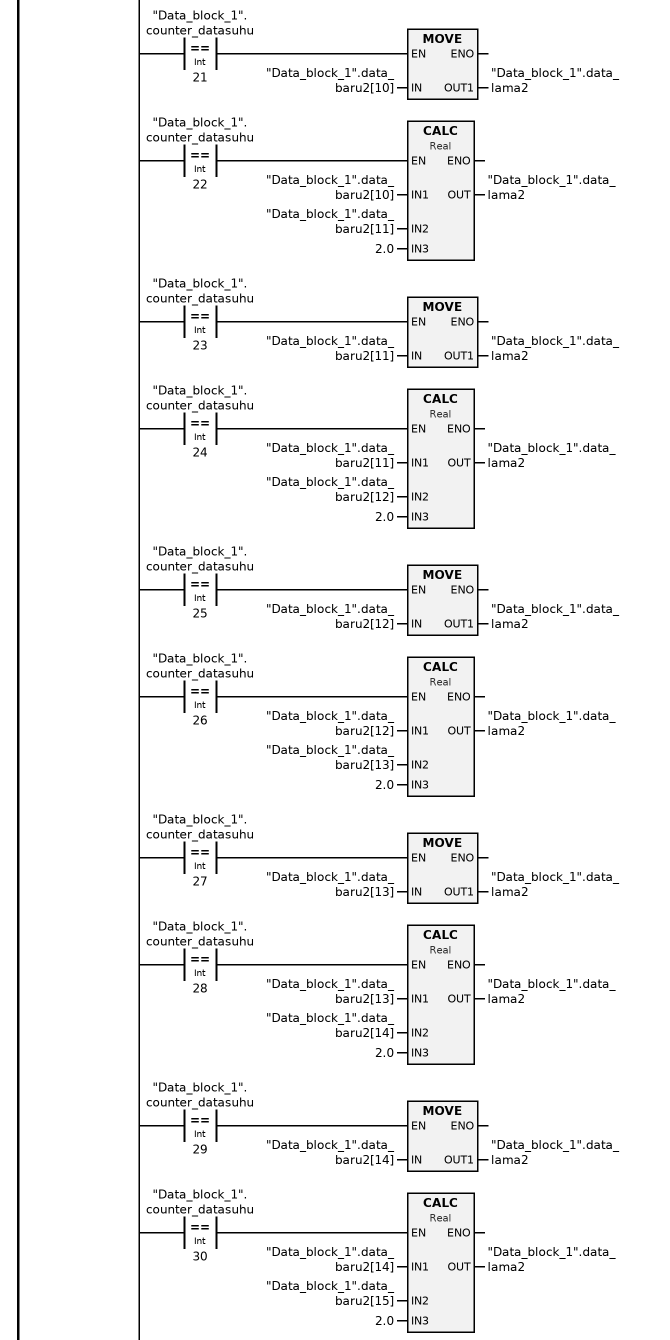
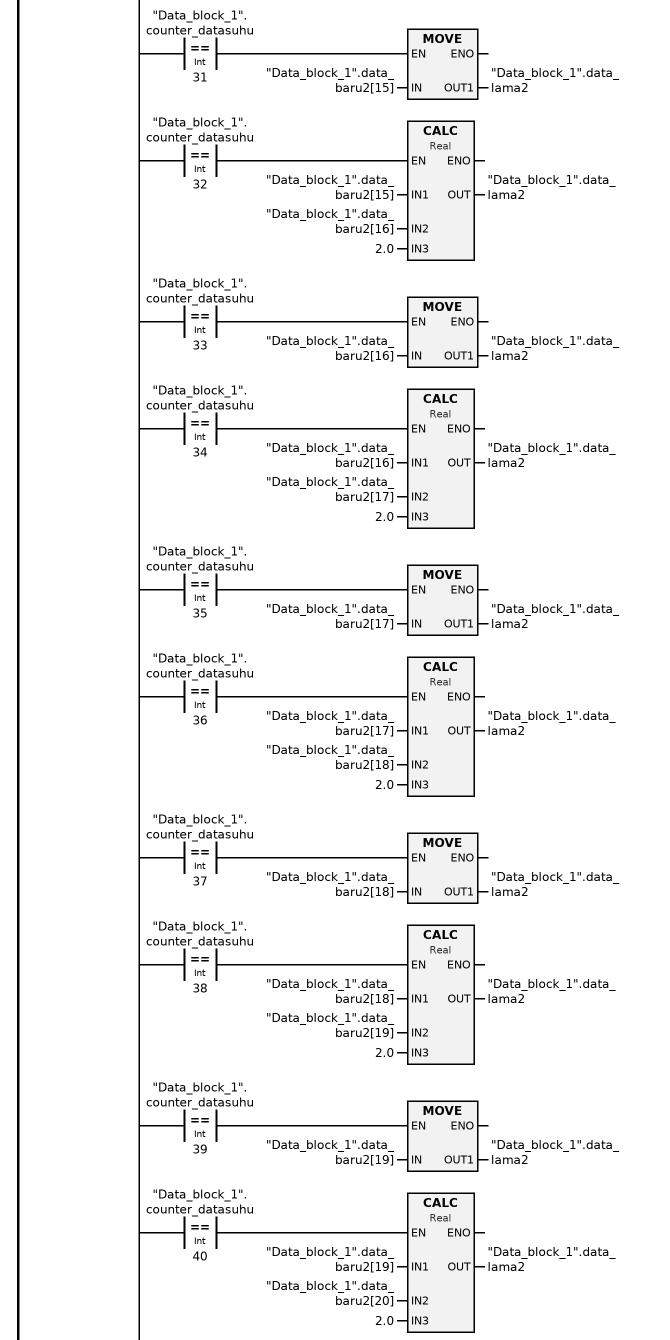
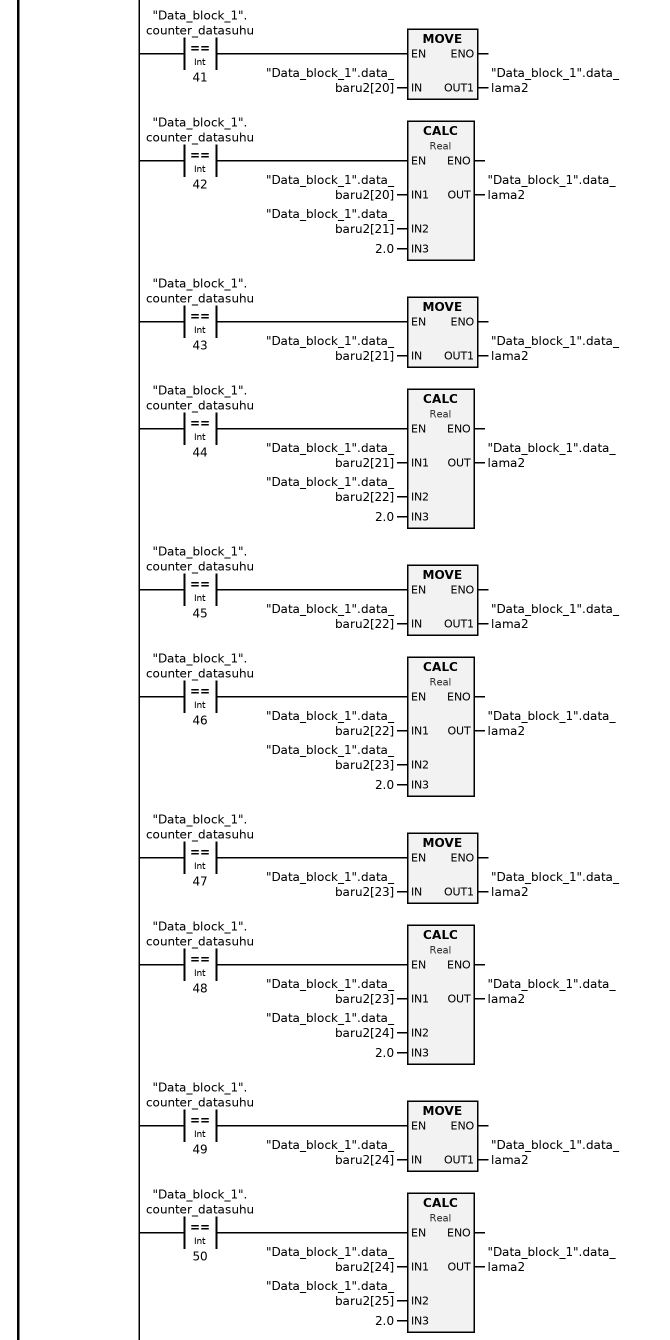
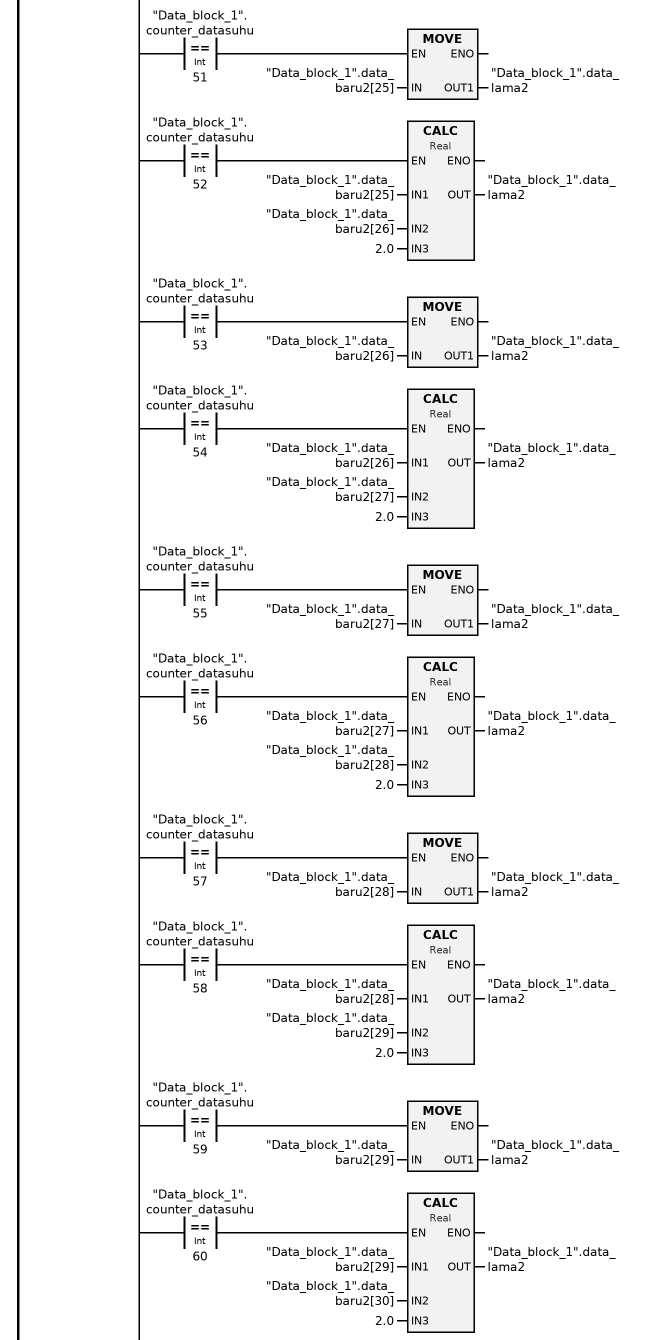
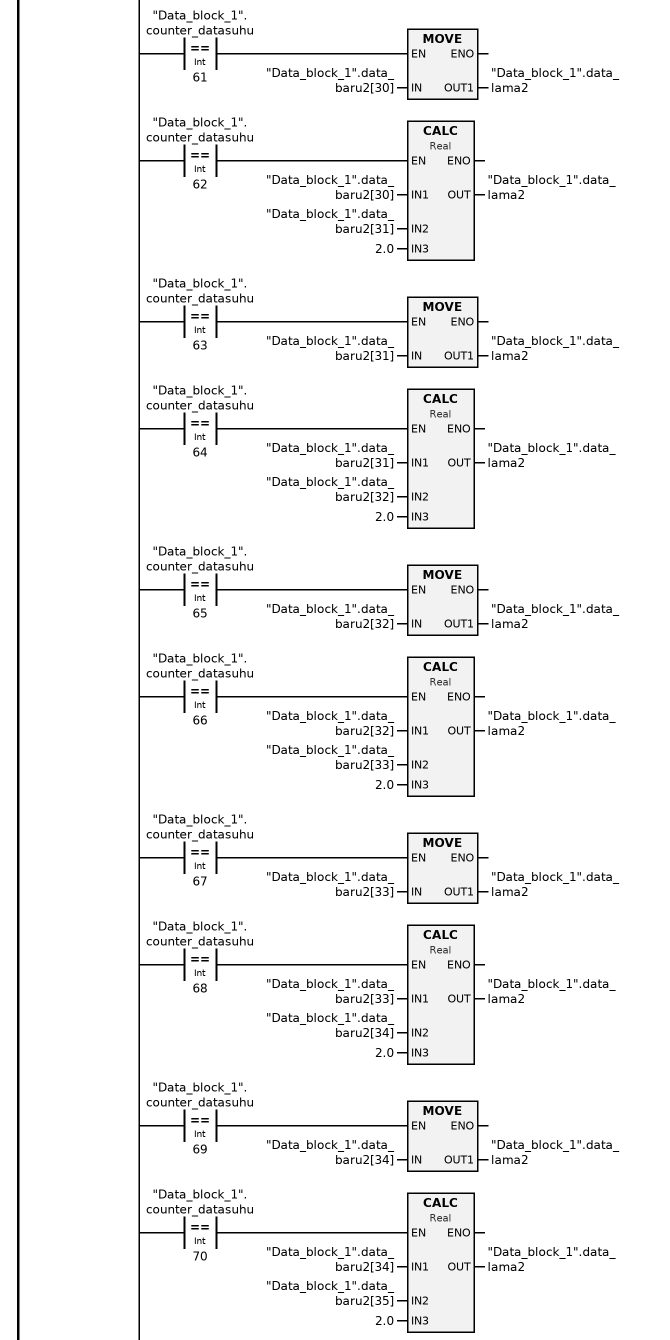
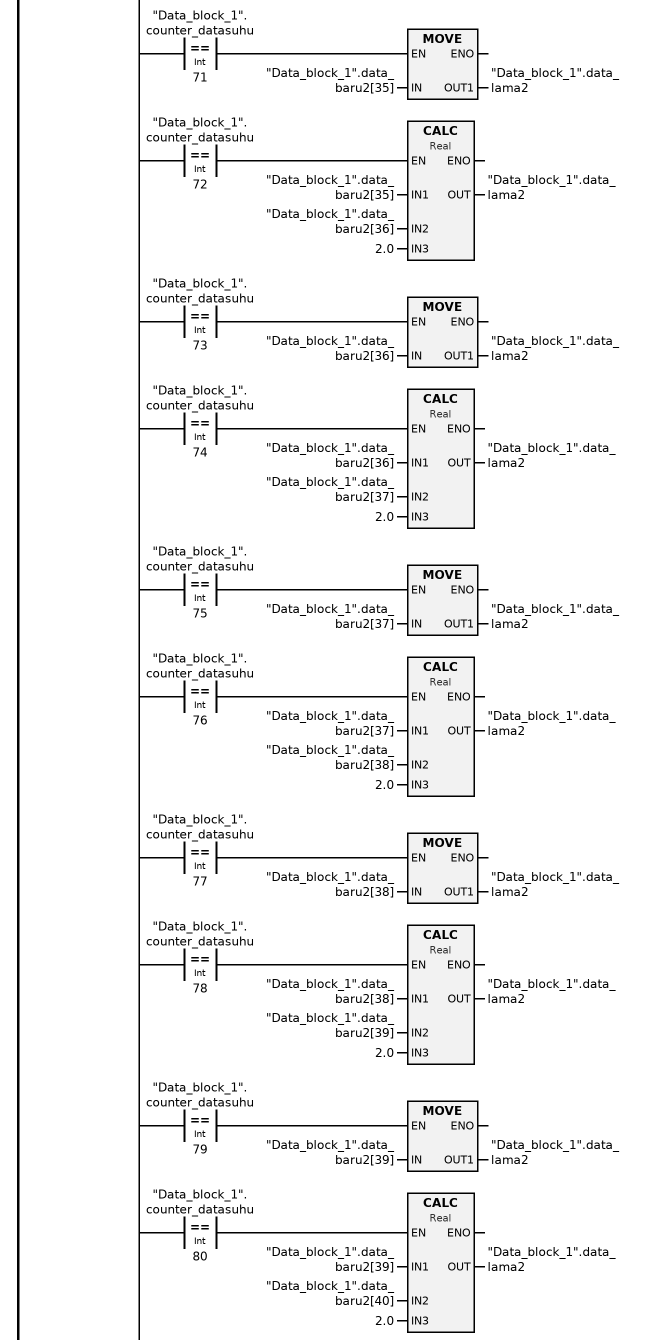
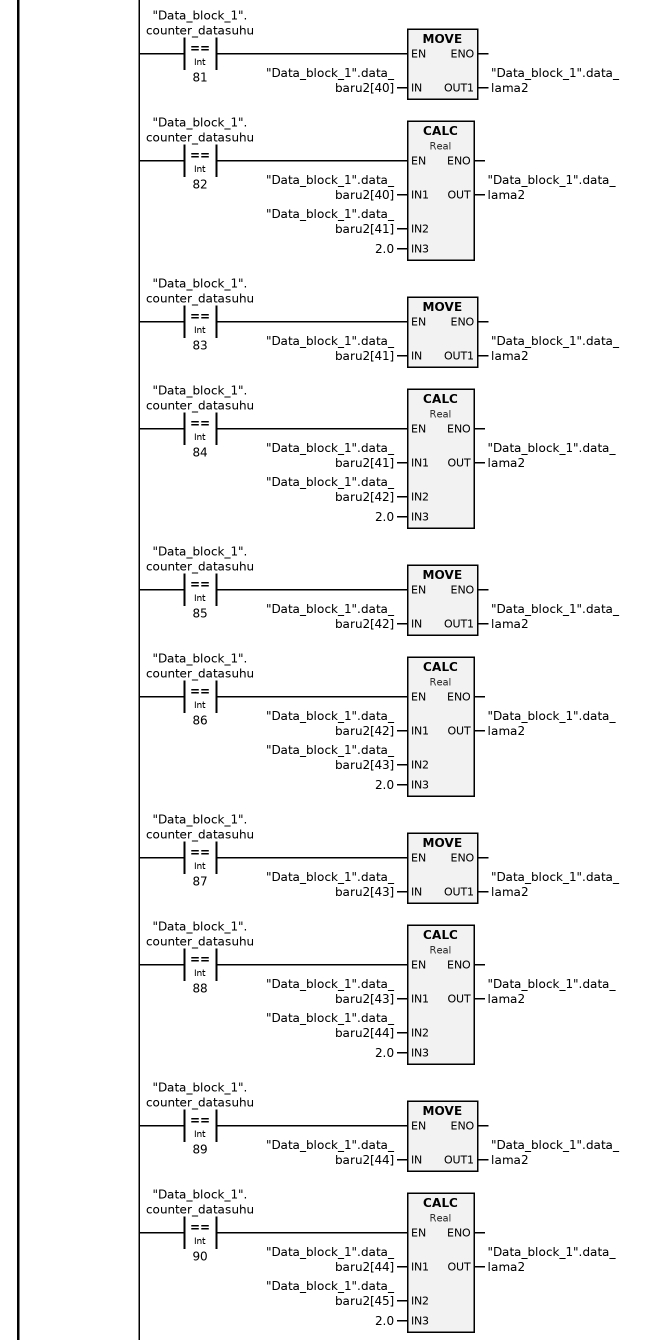
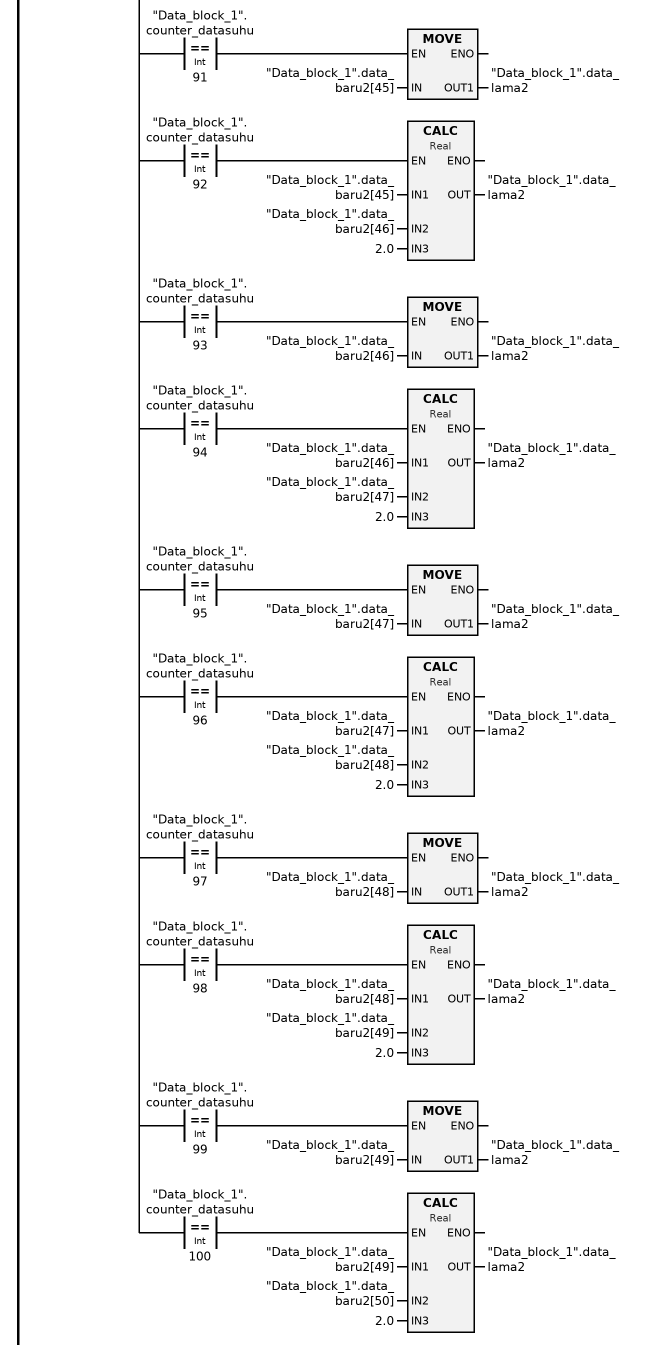
   #_w1 := NOT "Data_block_1".Lock_A;
   IF #_w1 AND ("Data_block_1".counter_datasuhu = 1) THEN
       "Data_block_1".data_lama2 := "Data_block_1".data_baru2[0];
   END_IF;
   IF #_w1 AND ("Data_block_1".counter_datasuhu = 2) THEN
       CALC(in1 := "Data_block_1".data_baru2[0],
            in2 := "Data_block_1".data_baru2[1],
            in3 := 2.0,
            out => "Data_block_1".data_lama2);
   END_IF;
   IF #_w1 AND ("Data_block_1".counter_datasuhu = 3) THEN
       "Data_block_1".data_lama2 := "Data_block_1".data_baru2[1];
   END_IF;
   IF #_w1 AND ("Data_block_1".counter_datasuhu = 4) THEN
       CALC(in1 := "Data_block_1".data_baru2[1],
            in2 := "Data_block_1".data_baru2[2],
            in3 := 2.0,
            out => "Data_block_1".data_lama2);
   END_IF;
   IF #_w1 AND ("Data_block_1".counter_datasuhu = 5) THEN
       "Data_block_1".data_lama2 := "Data_block_1".data_baru2[2];
   END_IF;
   IF #_w1 AND ("Data_block_1".counter_datasuhu = 6) THEN
       CALC(in1 := "Data_block_1".data_baru2[2],
            in2 := "Data_block_1".data_baru2[3],
            in3 := 2.0,
            out => "Data_block_1".data_lama2);
   END_IF;
   IF #_w1 AND ("Data_block_1".counter_datasuhu = 7) THEN
       "Data_block_1".data_lama2 := "Data_block_1".data_baru2[3];
   END_IF;
   IF #_w1 AND ("Data_block_1".counter_datasuhu = 8) THEN
       CALC(in1 := "Data_block_1".data_baru2[3],
            in2 := "Data_block_1".data_baru2[4],
            in3 := 2.0,
            out => "Data_block_1".data_lama2);
   END_IF;
   IF #_w1 AND ("Data_block_1".counter_datasuhu = 9) THEN
       "Data_block_1".data_lama2 := "Data_block_1".data_baru2[4];
   END_IF;
   IF #_w1 AND ("Data_block_1".counter_datasuhu = 10) THEN
       CALC(in1 := "Data_block_1".data_baru2[4],
            in2 := "Data_block_1".data_baru2[5],
            in3 := 2.0,
            out => "Data_block_1".data_lama2);
   END_IF;
   IF #_w1 AND ("Data_block_1".counter_datasuhu = 11) THEN
       "Data_block_1".data_lama2 := "Data_block_1".data_baru2[5];
   END_IF;
   IF #_w1 AND ("Data_block_1".counter_datasuhu = 12) THEN
       CALC(in1 := "Data_block_1".data_baru2[5],
            in2 := "Data_block_1".data_baru2[6],
            in3 := 2.0,
            out => "Data_block_1".data_lama2);
   END_IF;
   IF #_w1 AND ("Data_block_1".counter_datasuhu = 13) THEN
       "Data_block_1".data_lama2 := "Data_block_1".data_baru2[6];
   END_IF;
   IF #_w1 AND ("Data_block_1".counter_datasuhu = 14) THEN
       CALC(in1 := "Data_block_1".data_baru2[6],
            in2 := "Data_block_1".data_baru2[7],
            in3 := 2.0,
            out => "Data_block_1".data_lama2);
   END_IF;
   IF #_w1 AND ("Data_block_1".counter_datasuhu = 15) THEN
       "Data_block_1".data_lama2 := "Data_block_1".data_baru2[7];
   END_IF;
   IF #_w1 AND ("Data_block_1".counter_datasuhu = 16) THEN
       CALC(in1 := "Data_block_1".data_baru2[7],
            in2 := "Data_block_1".data_baru2[8],
            in3 := 2.0,
            out => "Data_block_1".data_lama2);
   END_IF;
   IF #_w1 AND ("Data_block_1".counter_datasuhu = 17) THEN
       "Data_block_1".data_lama2 := "Data_block_1".data_baru2[8];
   END_IF;
   IF #_w1 AND ("Data_block_1".counter_datasuhu = 18) THEN
       CALC(in1 := "Data_block_1".data_baru2[8],
            in2 := "Data_block_1".data_baru2[9],
            in3 := 2.0,
            out => "Data_block_1".data_lama2);
   END_IF;
   IF #_w1 AND ("Data_block_1".counter_datasuhu = 19) THEN
       "Data_block_1".data_lama2 := "Data_block_1".data_baru2[9];
   END_IF;
   IF #_w1 AND ("Data_block_1".counter_datasuhu = 20) THEN
       CALC(in1 := "Data_block_1".data_baru2[9],
            in2 := "Data_block_1".data_baru2[10],
            in3 := 2.0,
            out => "Data_block_1".data_lama2);
   END_IF;
   IF #_w1 AND ("Data_block_1".counter_datasuhu = 21) THEN
       "Data_block_1".data_lama2 := "Data_block_1".data_baru2[10];
   END_IF;
   IF #_w1 AND ("Data_block_1".counter_datasuhu = 22) THEN
       CALC(in1 := "Data_block_1".data_baru2[10],
            in2 := "Data_block_1".data_baru2[11],
            in3 := 2.0,
            out => "Data_block_1".data_lama2);
   END_IF;
   IF #_w1 AND ("Data_block_1".counter_datasuhu = 23) THEN
       "Data_block_1".data_lama2 := "Data_block_1".data_baru2[11];
   END_IF;
   IF #_w1 AND ("Data_block_1".counter_datasuhu = 24) THEN
       CALC(in1 := "Data_block_1".data_baru2[11],
            in2 := "Data_block_1".data_baru2[12],
            in3 := 2.0,
            out => "Data_block_1".data_lama2);
   END_IF;
   IF #_w1 AND ("Data_block_1".counter_datasuhu = 25) THEN
       "Data_block_1".data_lama2 := "Data_block_1".data_baru2[12];
   END_IF;
   IF #_w1 AND ("Data_block_1".counter_datasuhu = 26) THEN
       CALC(in1 := "Data_block_1".data_baru2[12],
            in2 := "Data_block_1".data_baru2[13],
            in3 := 2.0,
            out => "Data_block_1".data_lama2);
   END_IF;
   IF #_w1 AND ("Data_block_1".counter_datasuhu = 27) THEN
       "Data_block_1".data_lama2 := "Data_block_1".data_baru2[13];
   END_IF;
   IF #_w1 AND ("Data_block_1".counter_datasuhu = 28) THEN
       CALC(in1 := "Data_block_1".data_baru2[13],
            in2 := "Data_block_1".data_baru2[14],
            in3 := 2.0,
            out => "Data_block_1".data_lama2);
   END_IF;
   IF #_w1 AND ("Data_block_1".counter_datasuhu = 29) THEN
       "Data_block_1".data_lama2 := "Data_block_1".data_baru2[14];
   END_IF;
   IF #_w1 AND ("Data_block_1".counter_datasuhu = 30) THEN
       CALC(in1 := "Data_block_1".data_baru2[14],
            in2 := "Data_block_1".data_baru2[15],
            in3 := 2.0,
            out => "Data_block_1".data_lama2);
   END_IF;
   IF #_w1 AND ("Data_block_1".counter_datasuhu = 31) THEN
       "Data_block_1".data_lama2 := "Data_block_1".data_baru2[15];
   END_IF;
   IF #_w1 AND ("Data_block_1".counter_datasuhu = 32) THEN
       CALC(in1 := "Data_block_1".data_baru2[15],
            in2 := "Data_block_1".data_baru2[16],
            in3 := 2.0,
            out => "Data_block_1".data_lama2);
   END_IF;
   IF #_w1 AND ("Data_block_1".counter_datasuhu = 33) THEN
       "Data_block_1".data_lama2 := "Data_block_1".data_baru2[16];
   END_IF;
   IF #_w1 AND ("Data_block_1".counter_datasuhu = 34) THEN
       CALC(in1 := "Data_block_1".data_baru2[16],
            in2 := "Data_block_1".data_baru2[17],
            in3 := 2.0,
            out => "Data_block_1".data_lama2);
   END_IF;
   IF #_w1 AND ("Data_block_1".counter_datasuhu = 35) THEN
       "Data_block_1".data_lama2 := "Data_block_1".data_baru2[17];
   END_IF;
   IF #_w1 AND ("Data_block_1".counter_datasuhu = 36) THEN
       CALC(in1 := "Data_block_1".data_baru2[17],
            in2 := "Data_block_1".data_baru2[18],
            in3 := 2.0,
            out => "Data_block_1".data_lama2);
   END_IF;
   IF #_w1 AND ("Data_block_1".counter_datasuhu = 37) THEN
       "Data_block_1".data_lama2 := "Data_block_1".data_baru2[18];
   END_IF;
   IF #_w1 AND ("Data_block_1".counter_datasuhu = 38) THEN
       CALC(in1 := "Data_block_1".data_baru2[18],
            in2 := "Data_block_1".data_baru2[19],
            in3 := 2.0,
            out => "Data_block_1".data_lama2);
   END_IF;
   IF #_w1 AND ("Data_block_1".counter_datasuhu = 39) THEN
       "Data_block_1".data_lama2 := "Data_block_1".data_baru2[19];
   END_IF;
   IF #_w1 AND ("Data_block_1".counter_datasuhu = 40) THEN
       CALC(in1 := "Data_block_1".data_baru2[19],
            in2 := "Data_block_1".data_baru2[20],
            in3 := 2.0,
            out => "Data_block_1".data_lama2);
   END_IF;
   IF #_w1 AND ("Data_block_1".counter_datasuhu = 41) THEN
       "Data_block_1".data_lama2 := "Data_block_1".data_baru2[20];
   END_IF;
   IF #_w1 AND ("Data_block_1".counter_datasuhu = 42) THEN
       CALC(in1 := "Data_block_1".data_baru2[20],
            in2 := "Data_block_1".data_baru2[21],
            in3 := 2.0,
            out => "Data_block_1".data_lama2);
   END_IF;
   IF #_w1 AND ("Data_block_1".counter_datasuhu = 43) THEN
       "Data_block_1".data_lama2 := "Data_block_1".data_baru2[21];
   END_IF;
   IF #_w1 AND ("Data_block_1".counter_datasuhu = 44) THEN
       CALC(in1 := "Data_block_1".data_baru2[21],
            in2 := "Data_block_1".data_baru2[22],
            in3 := 2.0,
            out => "Data_block_1".data_lama2);
   END_IF;
   IF #_w1 AND ("Data_block_1".counter_datasuhu = 45) THEN
       "Data_block_1".data_lama2 := "Data_block_1".data_baru2[22];
   END_IF;
   IF #_w1 AND ("Data_block_1".counter_datasuhu = 46) THEN
       CALC(in1 := "Data_block_1".data_baru2[22],
            in2 := "Data_block_1".data_baru2[23],
            in3 := 2.0,
            out => "Data_block_1".data_lama2);
   END_IF;
   IF #_w1 AND ("Data_block_1".counter_datasuhu = 47) THEN
       "Data_block_1".data_lama2 := "Data_block_1".data_baru2[23];
   END_IF;
   IF #_w1 AND ("Data_block_1".counter_datasuhu = 48) THEN
       CALC(in1 := "Data_block_1".data_baru2[23],
            in2 := "Data_block_1".data_baru2[24],
            in3 := 2.0,
            out => "Data_block_1".data_lama2);
   END_IF;
   IF #_w1 AND ("Data_block_1".counter_datasuhu = 49) THEN
       "Data_block_1".data_lama2 := "Data_block_1".data_baru2[24];
   END_IF;
   IF #_w1 AND ("Data_block_1".counter_datasuhu = 50) THEN
       CALC(in1 := "Data_block_1".data_baru2[24],
            in2 := "Data_block_1".data_baru2[25],
            in3 := 2.0,
            out => "Data_block_1".data_lama2);
   END_IF;
   IF #_w1 AND ("Data_block_1".counter_datasuhu = 51) THEN
       "Data_block_1".data_lama2 := "Data_block_1".data_baru2[25];
   END_IF;
   IF #_w1 AND ("Data_block_1".counter_datasuhu = 52) THEN
       CALC(in1 := "Data_block_1".data_baru2[25],
            in2 := "Data_block_1".data_baru2[26],
            in3 := 2.0,
            out => "Data_block_1".data_lama2);
   END_IF;
   IF #_w1 AND ("Data_block_1".counter_datasuhu = 53) THEN
       "Data_block_1".data_lama2 := "Data_block_1".data_baru2[26];
   END_IF;
   IF #_w1 AND ("Data_block_1".counter_datasuhu = 54) THEN
       CALC(in1 := "Data_block_1".data_baru2[26],
            in2 := "Data_block_1".data_baru2[27],
            in3 := 2.0,
            out => "Data_block_1".data_lama2);
   END_IF;
   IF #_w1 AND ("Data_block_1".counter_datasuhu = 55) THEN
       "Data_block_1".data_lama2 := "Data_block_1".data_baru2[27];
   END_IF;
   IF #_w1 AND ("Data_block_1".counter_datasuhu = 56) THEN
       CALC(in1 := "Data_block_1".data_baru2[27],
            in2 := "Data_block_1".data_baru2[28],
            in3 := 2.0,
            out => "Data_block_1".data_lama2);
   END_IF;
   IF #_w1 AND ("Data_block_1".counter_datasuhu = 57) THEN
       "Data_block_1".data_lama2 := "Data_block_1".data_baru2[28];
   END_IF;
   IF #_w1 AND ("Data_block_1".counter_datasuhu = 58) THEN
       CALC(in1 := "Data_block_1".data_baru2[28],
            in2 := "Data_block_1".data_baru2[29],
            in3 := 2.0,
            out => "Data_block_1".data_lama2);
   END_IF;
   IF #_w1 AND ("Data_block_1".counter_datasuhu = 59) THEN
       "Data_block_1".data_lama2 := "Data_block_1".data_baru2[29];
   END_IF;
   IF #_w1 AND ("Data_block_1".counter_datasuhu = 60) THEN
       CALC(in1 := "Data_block_1".data_baru2[29],
            in2 := "Data_block_1".data_baru2[30],
            in3 := 2.0,
            out => "Data_block_1".data_lama2);
   END_IF;
   IF #_w1 AND ("Data_block_1".counter_datasuhu = 61) THEN
       "Data_block_1".data_lama2 := "Data_block_1".data_baru2[30];
   END_IF;
   IF #_w1 AND ("Data_block_1".counter_datasuhu = 62) THEN
       CALC(in1 := "Data_block_1".data_baru2[30],
            in2 := "Data_block_1".data_baru2[31],
            in3 := 2.0,
            out => "Data_block_1".data_lama2);
   END_IF;
   IF #_w1 AND ("Data_block_1".counter_datasuhu = 63) THEN
       "Data_block_1".data_lama2 := "Data_block_1".data_baru2[31];
   END_IF;
   IF #_w1 AND ("Data_block_1".counter_datasuhu = 64) THEN
       CALC(in1 := "Data_block_1".data_baru2[31],
            in2 := "Data_block_1".data_baru2[32],
            in3 := 2.0,
            out => "Data_block_1".data_lama2);
   END_IF;
   IF #_w1 AND ("Data_block_1".counter_datasuhu = 65) THEN
       "Data_block_1".data_lama2 := "Data_block_1".data_baru2[32];
   END_IF;
   IF #_w1 AND ("Data_block_1".counter_datasuhu = 66) THEN
       CALC(in1 := "Data_block_1".data_baru2[32],
            in2 := "Data_block_1".data_baru2[33],
            in3 := 2.0,
            out => "Data_block_1".data_lama2);
   END_IF;
   IF #_w1 AND ("Data_block_1".counter_datasuhu = 67) THEN
       "Data_block_1".data_lama2 := "Data_block_1".data_baru2[33];
   END_IF;
   IF #_w1 AND ("Data_block_1".counter_datasuhu = 68) THEN
       CALC(in1 := "Data_block_1".data_baru2[33],
            in2 := "Data_block_1".data_baru2[34],
            in3 := 2.0,
            out => "Data_block_1".data_lama2);
   END_IF;
   IF #_w1 AND ("Data_block_1".counter_datasuhu = 69) THEN
       "Data_block_1".data_lama2 := "Data_block_1".data_baru2[34];
   END_IF;
   IF #_w1 AND ("Data_block_1".counter_datasuhu = 70) THEN
       CALC(in1 := "Data_block_1".data_baru2[34],
            in2 := "Data_block_1".data_baru2[35],
            in3 := 2.0,
            out => "Data_block_1".data_lama2);
   END_IF;
   IF #_w1 AND ("Data_block_1".counter_datasuhu = 71) THEN
       "Data_block_1".data_lama2 := "Data_block_1".data_baru2[35];
   END_IF;
   IF #_w1 AND ("Data_block_1".counter_datasuhu = 72) THEN
       CALC(in1 := "Data_block_1".data_baru2[35],
            in2 := "Data_block_1".data_baru2[36],
            in3 := 2.0,
            out => "Data_block_1".data_lama2);
   END_IF;
   IF #_w1 AND ("Data_block_1".counter_datasuhu = 73) THEN
       "Data_block_1".data_lama2 := "Data_block_1".data_baru2[36];
   END_IF;
   IF #_w1 AND ("Data_block_1".counter_datasuhu = 74) THEN
       CALC(in1 := "Data_block_1".data_baru2[36],
            in2 := "Data_block_1".data_baru2[37],
            in3 := 2.0,
            out => "Data_block_1".data_lama2);
   END_IF;
   IF #_w1 AND ("Data_block_1".counter_datasuhu = 75) THEN
       "Data_block_1".data_lama2 := "Data_block_1".data_baru2[37];
   END_IF;
   IF #_w1 AND ("Data_block_1".counter_datasuhu = 76) THEN
       CALC(in1 := "Data_block_1".data_baru2[37],
            in2 := "Data_block_1".data_baru2[38],
            in3 := 2.0,
            out => "Data_block_1".data_lama2);
   END_IF;
   IF #_w1 AND ("Data_block_1".counter_datasuhu = 77) THEN
       "Data_block_1".data_lama2 := "Data_block_1".data_baru2[38];
   END_IF;
   IF #_w1 AND ("Data_block_1".counter_datasuhu = 78) THEN
       CALC(in1 := "Data_block_1".data_baru2[38],
            in2 := "Data_block_1".data_baru2[39],
            in3 := 2.0,
            out => "Data_block_1".data_lama2);
   END_IF;
   IF #_w1 AND ("Data_block_1".counter_datasuhu = 79) THEN
       "Data_block_1".data_lama2 := "Data_block_1".data_baru2[39];
   END_IF;
   IF #_w1 AND ("Data_block_1".counter_datasuhu = 80) THEN
       CALC(in1 := "Data_block_1".data_baru2[39],
            in2 := "Data_block_1".data_baru2[40],
            in3 := 2.0,
            out => "Data_block_1".data_lama2);
   END_IF;
   IF #_w1 AND ("Data_block_1".counter_datasuhu = 81) THEN
       "Data_block_1".data_lama2 := "Data_block_1".data_baru2[40];
   END_IF;
   IF #_w1 AND ("Data_block_1".counter_datasuhu = 82) THEN
       CALC(in1 := "Data_block_1".data_baru2[40],
            in2 := "Data_block_1".data_baru2[41],
            in3 := 2.0,
            out => "Data_block_1".data_lama2);
   END_IF;
   IF #_w1 AND ("Data_block_1".counter_datasuhu = 83) THEN
       "Data_block_1".data_lama2 := "Data_block_1".data_baru2[41];
   END_IF;
   IF #_w1 AND ("Data_block_1".counter_datasuhu = 84) THEN
       CALC(in1 := "Data_block_1".data_baru2[41],
            in2 := "Data_block_1".data_baru2[42],
            in3 := 2.0,
            out => "Data_block_1".data_lama2);
   END_IF;
   IF #_w1 AND ("Data_block_1".counter_datasuhu = 85) THEN
       "Data_block_1".data_lama2 := "Data_block_1".data_baru2[42];
   END_IF;
   IF #_w1 AND ("Data_block_1".counter_datasuhu = 86) THEN
       CALC(in1 := "Data_block_1".data_baru2[42],
            in2 := "Data_block_1".data_baru2[43],
            in3 := 2.0,
            out => "Data_block_1".data_lama2);
   END_IF;
   IF #_w1 AND ("Data_block_1".counter_datasuhu = 87) THEN
       "Data_block_1".data_lama2 := "Data_block_1".data_baru2[43];
   END_IF;
   IF #_w1 AND ("Data_block_1".counter_datasuhu = 88) THEN
       CALC(in1 := "Data_block_1".data_baru2[43],
            in2 := "Data_block_1".data_baru2[44],
            in3 := 2.0,
            out => "Data_block_1".data_lama2);
   END_IF;
   IF #_w1 AND ("Data_block_1".counter_datasuhu = 89) THEN
       "Data_block_1".data_lama2 := "Data_block_1".data_baru2[44];
   END_IF;
   IF #_w1 AND ("Data_block_1".counter_datasuhu = 90) THEN
       CALC(in1 := "Data_block_1".data_baru2[44],
            in2 := "Data_block_1".data_baru2[45],
            in3 := 2.0,
            out => "Data_block_1".data_lama2);
   END_IF;
   IF #_w1 AND ("Data_block_1".counter_datasuhu = 91) THEN
       "Data_block_1".data_lama2 := "Data_block_1".data_baru2[45];
   END_IF;
   IF #_w1 AND ("Data_block_1".counter_datasuhu = 92) THEN
       CALC(in1 := "Data_block_1".data_baru2[45],
            in2 := "Data_block_1".data_baru2[46],
            in3 := 2.0,
            out => "Data_block_1".data_lama2);
   END_IF;
   IF #_w1 AND ("Data_block_1".counter_datasuhu = 93) THEN
       "Data_block_1".data_lama2 := "Data_block_1".data_baru2[46];
   END_IF;
   IF #_w1 AND ("Data_block_1".counter_datasuhu = 94) THEN
       CALC(in1 := "Data_block_1".data_baru2[46],
            in2 := "Data_block_1".data_baru2[47],
            in3 := 2.0,
            out => "Data_block_1".data_lama2);
   END_IF;
   IF #_w1 AND ("Data_block_1".counter_datasuhu = 95) THEN
       "Data_block_1".data_lama2 := "Data_block_1".data_baru2[47];
   END_IF;
   IF #_w1 AND ("Data_block_1".counter_datasuhu = 96) THEN
       CALC(in1 := "Data_block_1".data_baru2[47],
            in2 := "Data_block_1".data_baru2[48],
            in3 := 2.0,
            out => "Data_block_1".data_lama2);
   END_IF;
   IF #_w1 AND ("Data_block_1".counter_datasuhu = 97) THEN
       "Data_block_1".data_lama2 := "Data_block_1".data_baru2[48];
   END_IF;
   IF #_w1 AND ("Data_block_1".counter_datasuhu = 98) THEN
       CALC(in1 := "Data_block_1".data_baru2[48],
            in2 := "Data_block_1".data_baru2[49],
            in3 := 2.0,
            out => "Data_block_1".data_lama2);
   END_IF;
   IF #_w1 AND ("Data_block_1".counter_datasuhu = 99) THEN
       "Data_block_1".data_lama2 := "Data_block_1".data_baru2[49];
   END_IF;
   IF #_w1 AND ("Data_block_1".counter_datasuhu = 100) THEN
       CALC(in1 := "Data_block_1".data_baru2[49],
            in2 := "Data_block_1".data_baru2[50],
            in3 := 2.0,
            out => "Data_block_1".data_lama2);
   END_IF;
END_REGION

REGION Network 29: Memasukkan Data
   // ketika pemutus aktif dan counter bertambah, data suhu lama dipindahkan ke array dataroda (dari 0-37) serta sarana akan ditampilkan pada tabel sesuai roda pertama tiap sarana
   // ketika pemutus aktif, data suhu, data suhu lama , dan data suhu baru akan menjadi 0
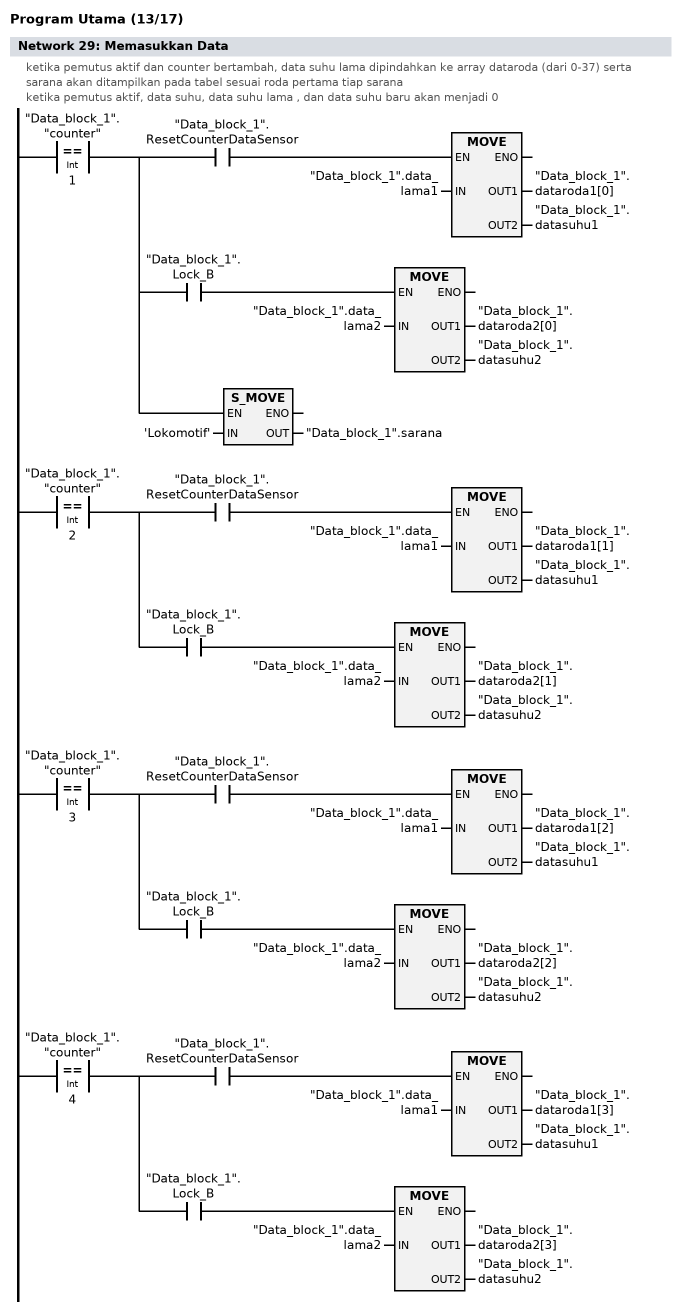
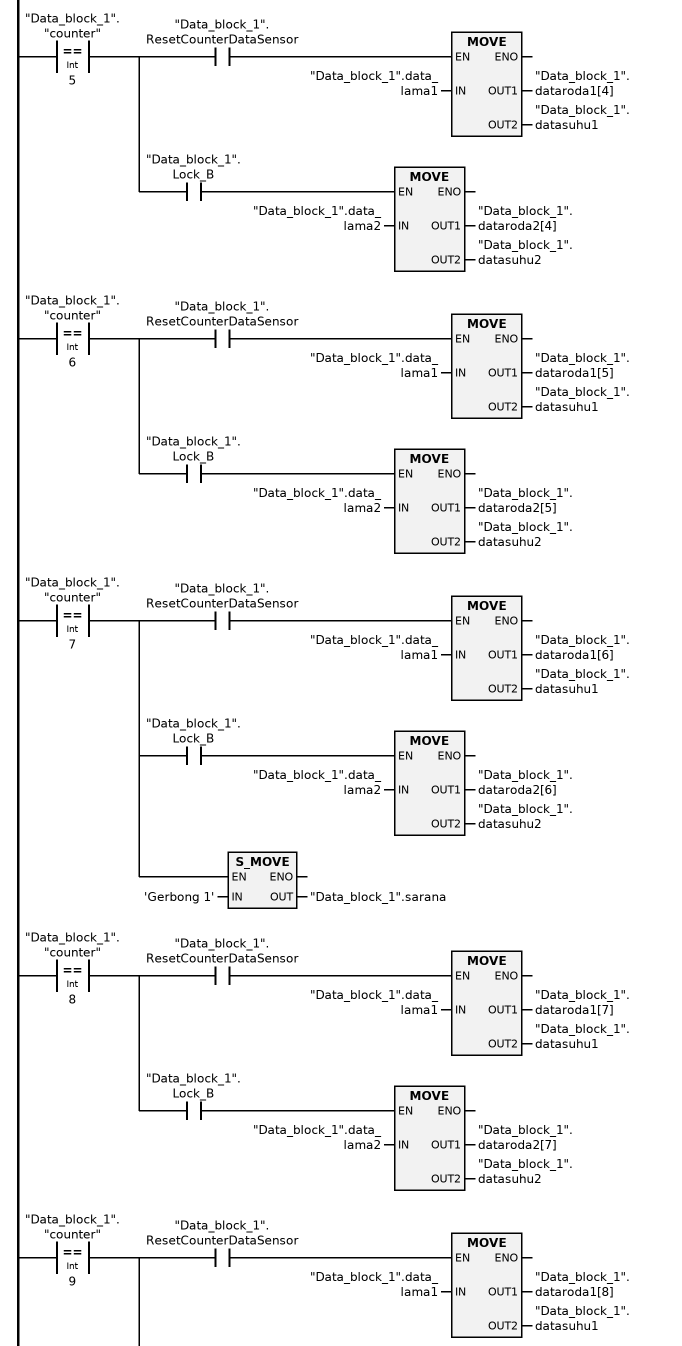
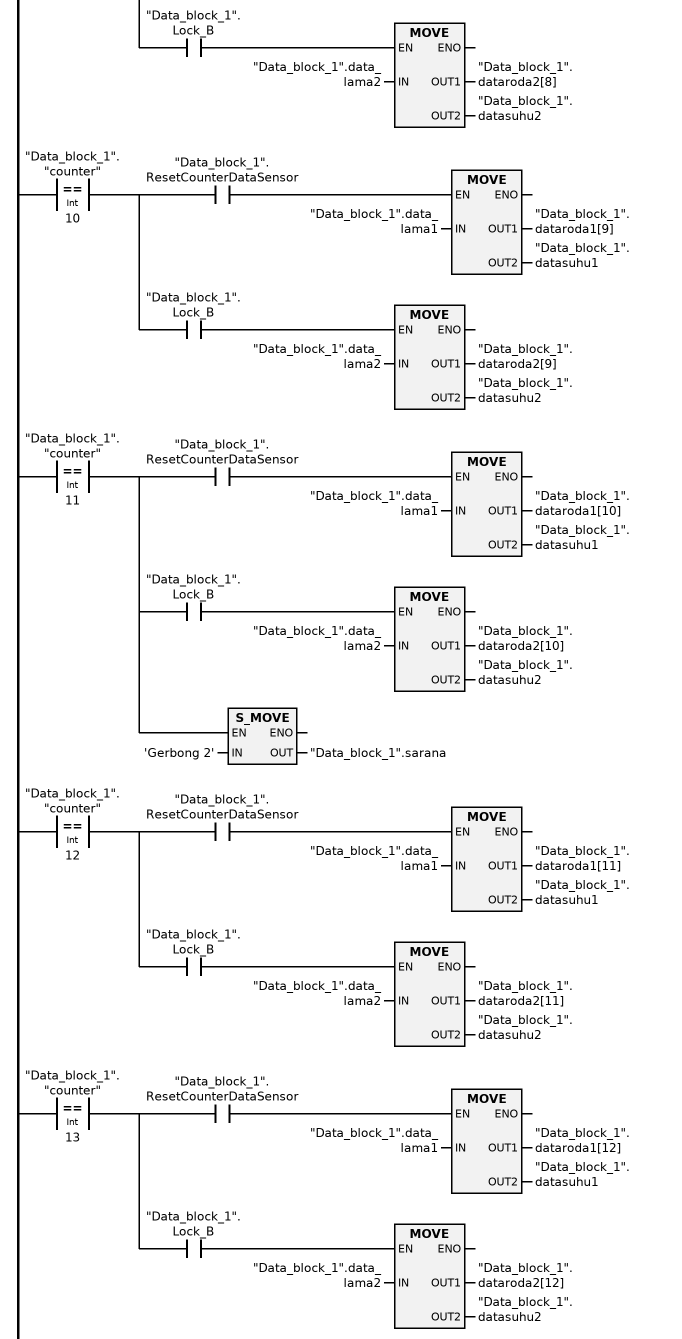
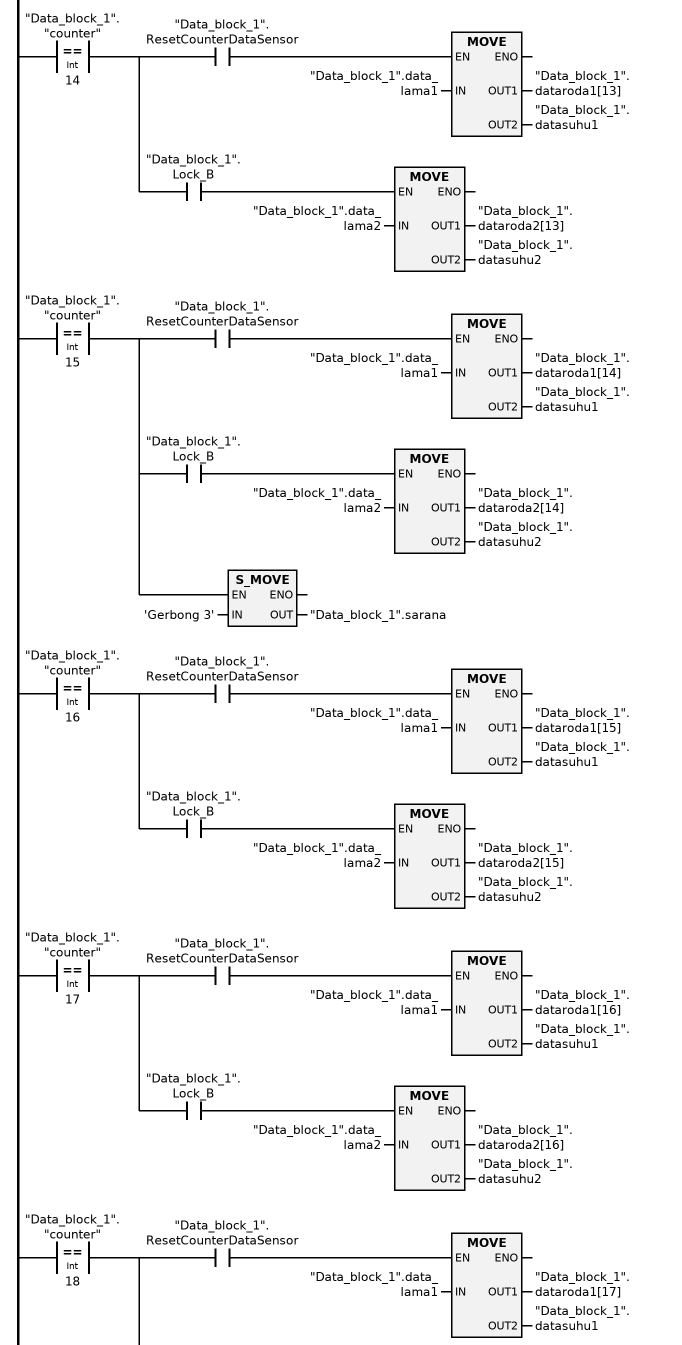
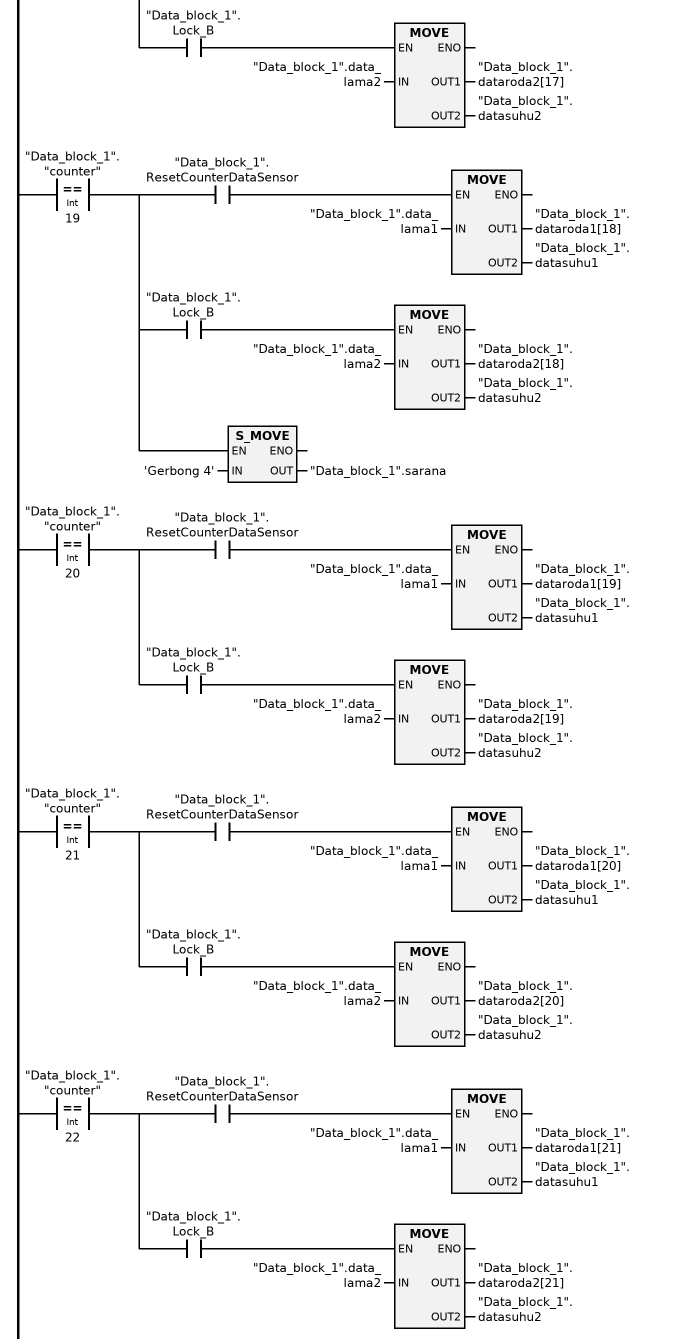
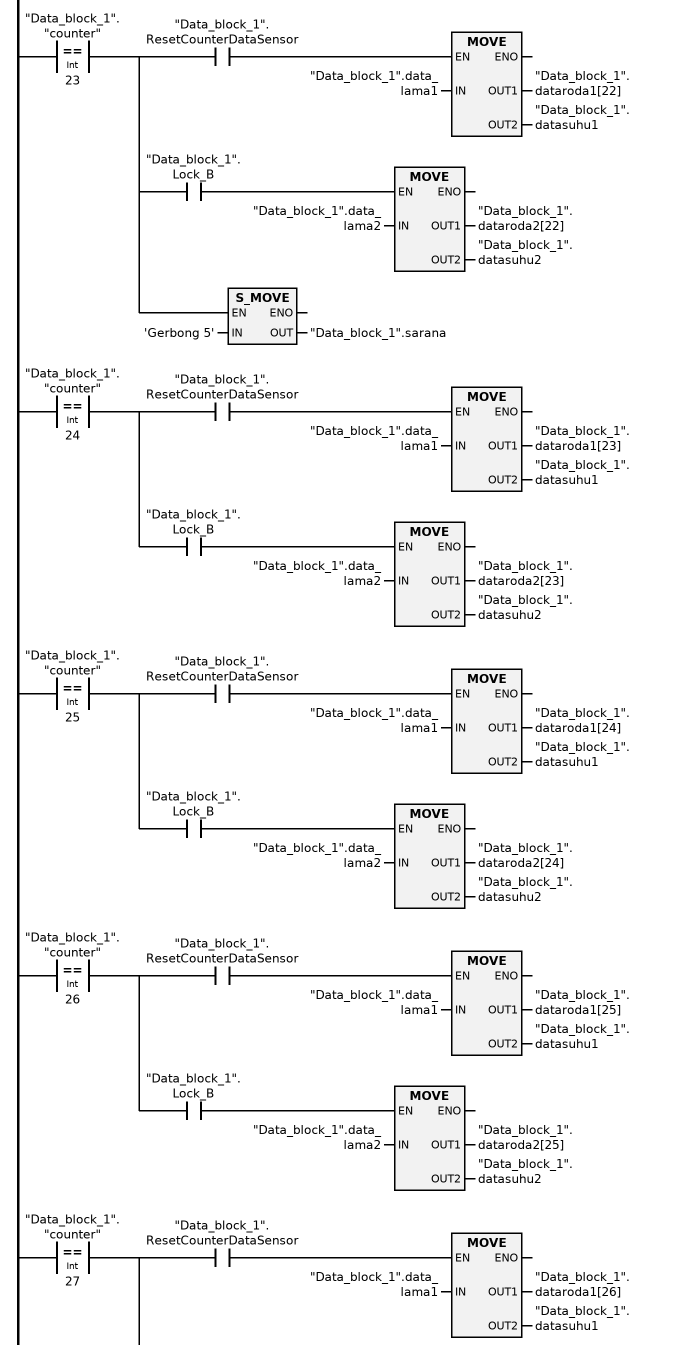
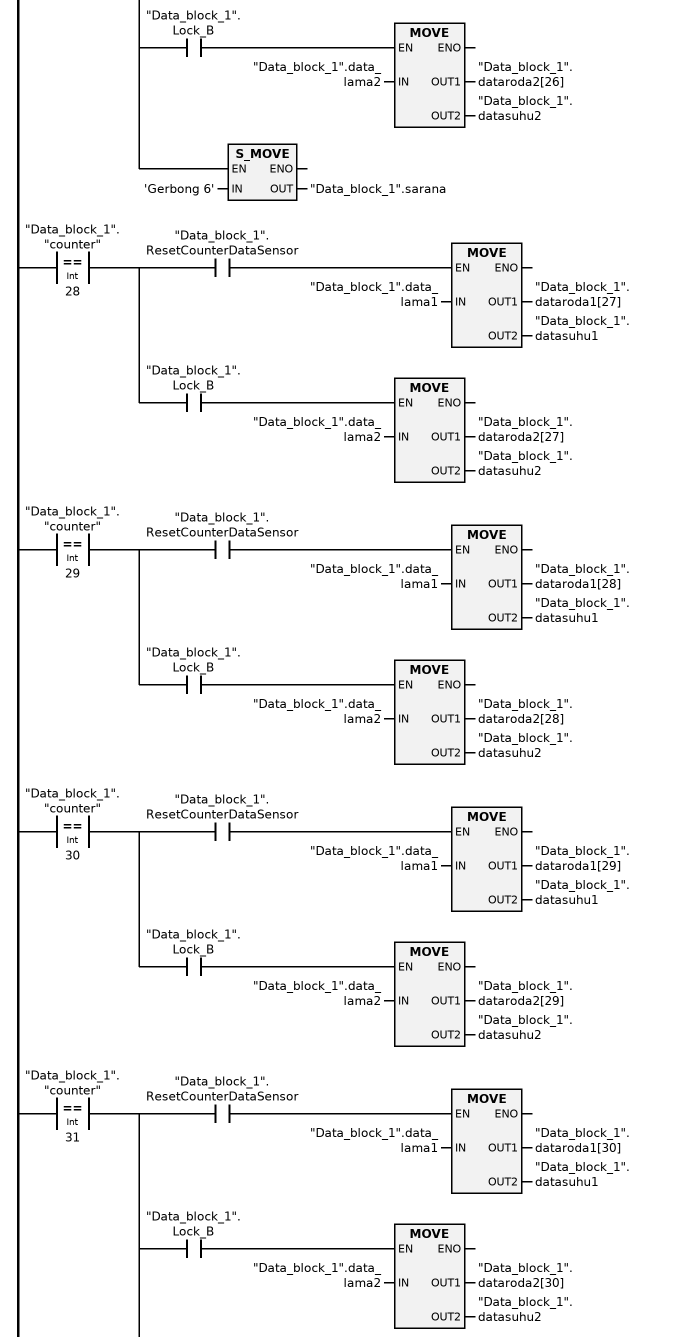
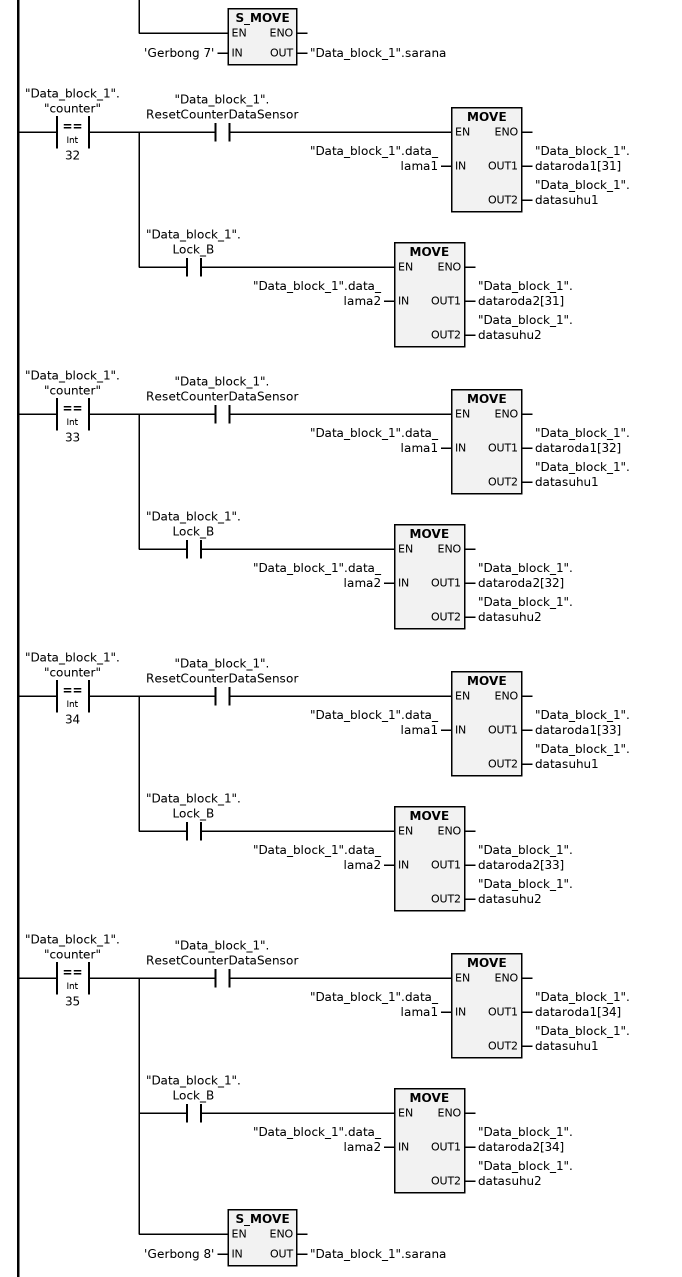
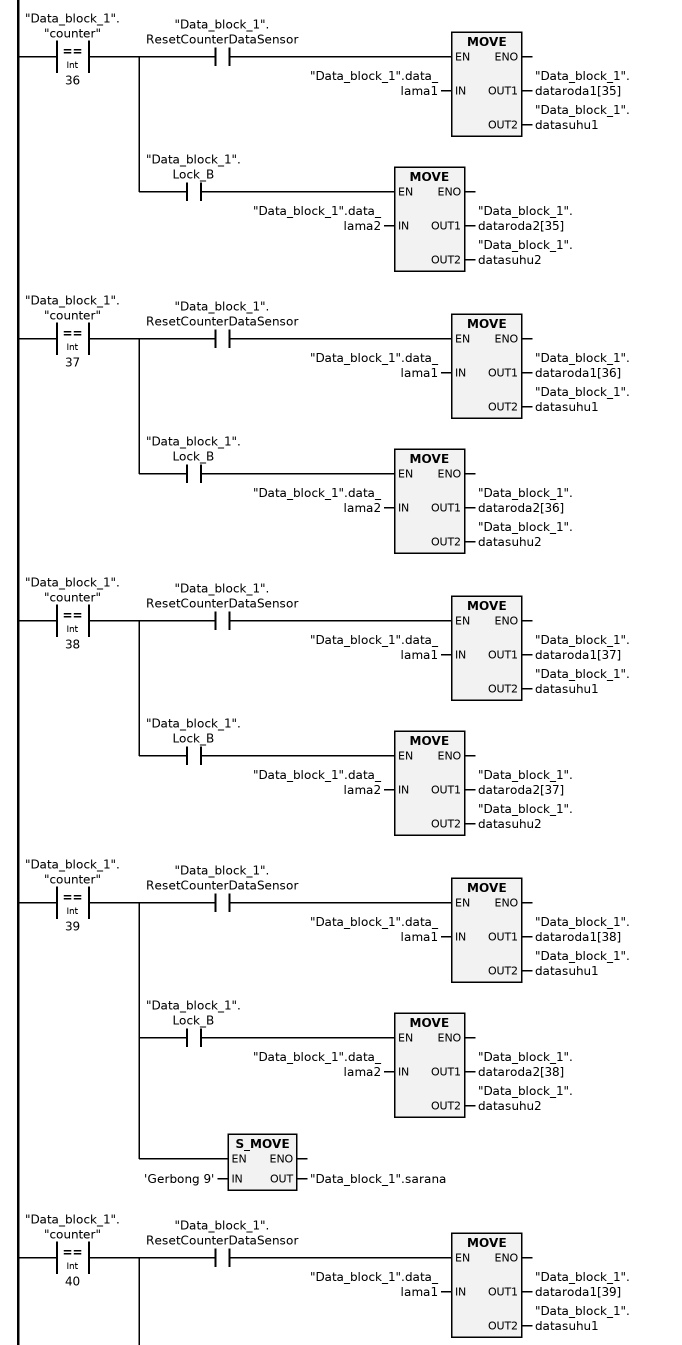
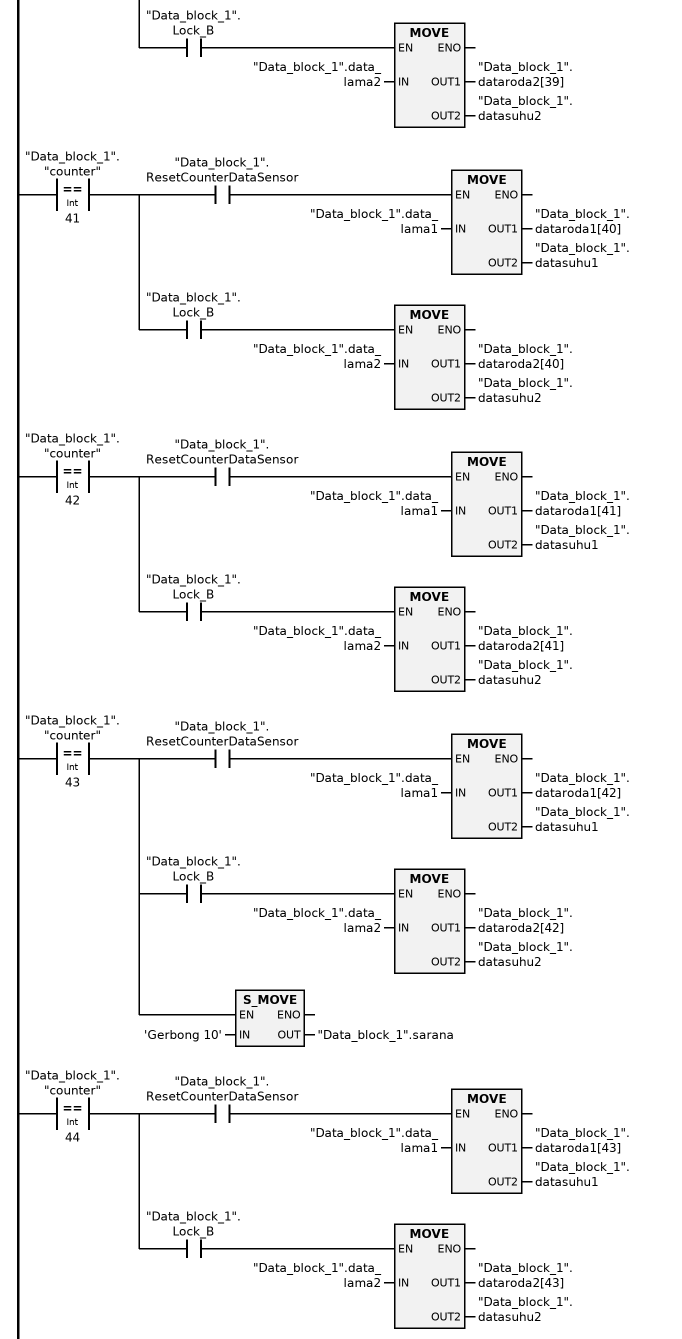
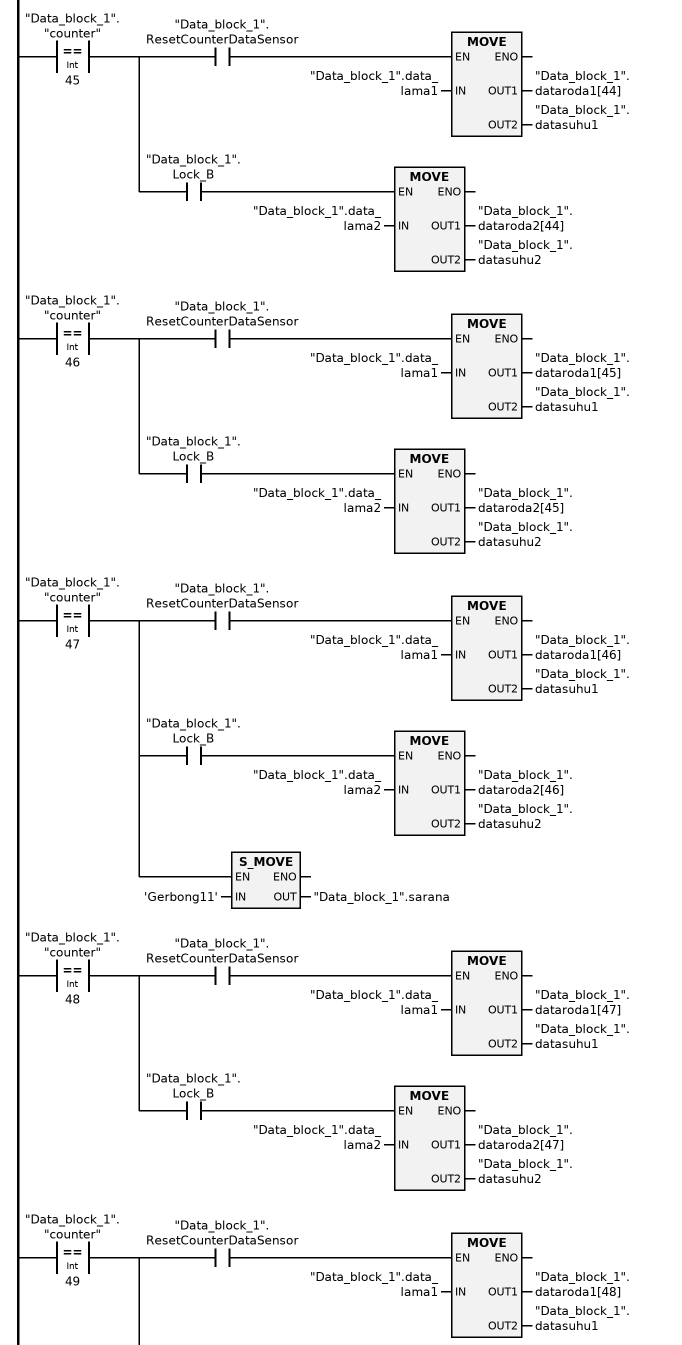
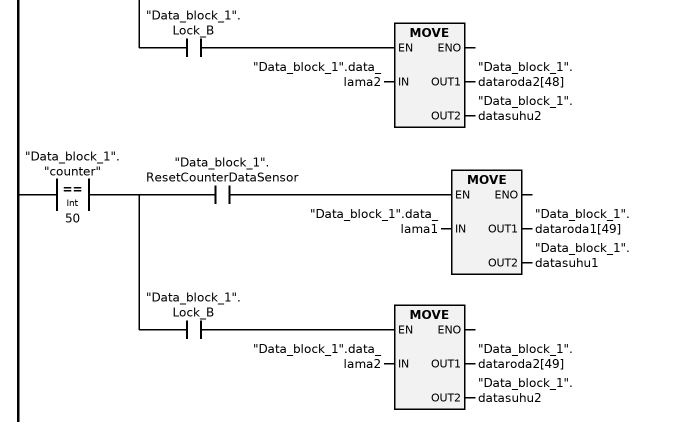
   #_w1 := "Data_block_1"."counter" = 1;
   IF #_w1 AND "Data_block_1".ResetCounterDataSensor THEN
       "Data_block_1".dataroda1[0] := "Data_block_1".data_lama1;
       "Data_block_1".datasuhu1 := "Data_block_1".data_lama1;
   END_IF;
   IF #_w1 AND "Data_block_1".Lock_B THEN
       "Data_block_1".dataroda2[0] := "Data_block_1".data_lama2;
       "Data_block_1".datasuhu2 := "Data_block_1".data_lama2;
   END_IF;
   IF #_w1 THEN S_MOVE(in := 'Lokomotif', out => "Data_block_1".sarana); END_IF;
   #_w2 := "Data_block_1"."counter" = 2;
   IF #_w2 AND "Data_block_1".ResetCounterDataSensor THEN
       "Data_block_1".dataroda1[1] := "Data_block_1".data_lama1;
       "Data_block_1".datasuhu1 := "Data_block_1".data_lama1;
   END_IF;
   IF #_w2 AND "Data_block_1".Lock_B THEN
       "Data_block_1".dataroda2[1] := "Data_block_1".data_lama2;
       "Data_block_1".datasuhu2 := "Data_block_1".data_lama2;
   END_IF;
   #_w3 := "Data_block_1"."counter" = 3;
   IF #_w3 AND "Data_block_1".ResetCounterDataSensor THEN
       "Data_block_1".dataroda1[2] := "Data_block_1".data_lama1;
       "Data_block_1".datasuhu1 := "Data_block_1".data_lama1;
   END_IF;
   IF #_w3 AND "Data_block_1".Lock_B THEN
       "Data_block_1".dataroda2[2] := "Data_block_1".data_lama2;
       "Data_block_1".datasuhu2 := "Data_block_1".data_lama2;
   END_IF;
   #_w4 := "Data_block_1"."counter" = 4;
   IF #_w4 AND "Data_block_1".ResetCounterDataSensor THEN
       "Data_block_1".dataroda1[3] := "Data_block_1".data_lama1;
       "Data_block_1".datasuhu1 := "Data_block_1".data_lama1;
   END_IF;
   IF #_w4 AND "Data_block_1".Lock_B THEN
       "Data_block_1".dataroda2[3] := "Data_block_1".data_lama2;
       "Data_block_1".datasuhu2 := "Data_block_1".data_lama2;
   END_IF;
   #_w5 := "Data_block_1"."counter" = 5;
   IF #_w5 AND "Data_block_1".ResetCounterDataSensor THEN
       "Data_block_1".dataroda1[4] := "Data_block_1".data_lama1;
       "Data_block_1".datasuhu1 := "Data_block_1".data_lama1;
   END_IF;
   IF #_w5 AND "Data_block_1".Lock_B THEN
       "Data_block_1".dataroda2[4] := "Data_block_1".data_lama2;
       "Data_block_1".datasuhu2 := "Data_block_1".data_lama2;
   END_IF;
   #_w6 := "Data_block_1"."counter" = 6;
   IF #_w6 AND "Data_block_1".ResetCounterDataSensor THEN
       "Data_block_1".dataroda1[5] := "Data_block_1".data_lama1;
       "Data_block_1".datasuhu1 := "Data_block_1".data_lama1;
   END_IF;
   IF #_w6 AND "Data_block_1".Lock_B THEN
       "Data_block_1".dataroda2[5] := "Data_block_1".data_lama2;
       "Data_block_1".datasuhu2 := "Data_block_1".data_lama2;
   END_IF;
   #_w7 := "Data_block_1"."counter" = 7;
   IF #_w7 AND "Data_block_1".ResetCounterDataSensor THEN
       "Data_block_1".dataroda1[6] := "Data_block_1".data_lama1;
       "Data_block_1".datasuhu1 := "Data_block_1".data_lama1;
   END_IF;
   IF #_w7 AND "Data_block_1".Lock_B THEN
       "Data_block_1".dataroda2[6] := "Data_block_1".data_lama2;
       "Data_block_1".datasuhu2 := "Data_block_1".data_lama2;
   END_IF;
   IF #_w7 THEN S_MOVE(in := 'Gerbong 1', out => "Data_block_1".sarana); END_IF;
   #_w8 := "Data_block_1"."counter" = 8;
   IF #_w8 AND "Data_block_1".ResetCounterDataSensor THEN
       "Data_block_1".dataroda1[7] := "Data_block_1".data_lama1;
       "Data_block_1".datasuhu1 := "Data_block_1".data_lama1;
   END_IF;
   IF #_w8 AND "Data_block_1".Lock_B THEN
       "Data_block_1".dataroda2[7] := "Data_block_1".data_lama2;
       "Data_block_1".datasuhu2 := "Data_block_1".data_lama2;
   END_IF;
   #_w9 := "Data_block_1"."counter" = 9;
   IF #_w9 AND "Data_block_1".ResetCounterDataSensor THEN
       "Data_block_1".dataroda1[8] := "Data_block_1".data_lama1;
       "Data_block_1".datasuhu1 := "Data_block_1".data_lama1;
   END_IF;
   IF #_w9 AND "Data_block_1".Lock_B THEN
       "Data_block_1".dataroda2[8] := "Data_block_1".data_lama2;
       "Data_block_1".datasuhu2 := "Data_block_1".data_lama2;
   END_IF;
   #_w10 := "Data_block_1"."counter" = 10;
   IF #_w10 AND "Data_block_1".ResetCounterDataSensor THEN
       "Data_block_1".dataroda1[9] := "Data_block_1".data_lama1;
       "Data_block_1".datasuhu1 := "Data_block_1".data_lama1;
   END_IF;
   IF #_w10 AND "Data_block_1".Lock_B THEN
       "Data_block_1".dataroda2[9] := "Data_block_1".data_lama2;
       "Data_block_1".datasuhu2 := "Data_block_1".data_lama2;
   END_IF;
   #_w11 := "Data_block_1"."counter" = 11;
   IF #_w11 AND "Data_block_1".ResetCounterDataSensor THEN
       "Data_block_1".dataroda1[10] := "Data_block_1".data_lama1;
       "Data_block_1".datasuhu1 := "Data_block_1".data_lama1;
   END_IF;
   IF #_w11 AND "Data_block_1".Lock_B THEN
       "Data_block_1".dataroda2[10] := "Data_block_1".data_lama2;
       "Data_block_1".datasuhu2 := "Data_block_1".data_lama2;
   END_IF;
   IF #_w11 THEN S_MOVE(in := 'Gerbong 2', out => "Data_block_1".sarana); END_IF;
   #_w12 := "Data_block_1"."counter" = 12;
   IF #_w12 AND "Data_block_1".ResetCounterDataSensor THEN
       "Data_block_1".dataroda1[11] := "Data_block_1".data_lama1;
       "Data_block_1".datasuhu1 := "Data_block_1".data_lama1;
   END_IF;
   IF #_w12 AND "Data_block_1".Lock_B THEN
       "Data_block_1".dataroda2[11] := "Data_block_1".data_lama2;
       "Data_block_1".datasuhu2 := "Data_block_1".data_lama2;
   END_IF;
   #_w13 := "Data_block_1"."counter" = 13;
   IF #_w13 AND "Data_block_1".ResetCounterDataSensor THEN
       "Data_block_1".dataroda1[12] := "Data_block_1".data_lama1;
       "Data_block_1".datasuhu1 := "Data_block_1".data_lama1;
   END_IF;
   IF #_w13 AND "Data_block_1".Lock_B THEN
       "Data_block_1".dataroda2[12] := "Data_block_1".data_lama2;
       "Data_block_1".datasuhu2 := "Data_block_1".data_lama2;
   END_IF;
   #_w14 := "Data_block_1"."counter" = 14;
   IF #_w14 AND "Data_block_1".ResetCounterDataSensor THEN
       "Data_block_1".dataroda1[13] := "Data_block_1".data_lama1;
       "Data_block_1".datasuhu1 := "Data_block_1".data_lama1;
   END_IF;
   IF #_w14 AND "Data_block_1".Lock_B THEN
       "Data_block_1".dataroda2[13] := "Data_block_1".data_lama2;
       "Data_block_1".datasuhu2 := "Data_block_1".data_lama2;
   END_IF;
   #_w15 := "Data_block_1"."counter" = 15;
   IF #_w15 AND "Data_block_1".ResetCounterDataSensor THEN
       "Data_block_1".dataroda1[14] := "Data_block_1".data_lama1;
       "Data_block_1".datasuhu1 := "Data_block_1".data_lama1;
   END_IF;
   IF #_w15 AND "Data_block_1".Lock_B THEN
       "Data_block_1".dataroda2[14] := "Data_block_1".data_lama2;
       "Data_block_1".datasuhu2 := "Data_block_1".data_lama2;
   END_IF;
   IF #_w15 THEN S_MOVE(in := 'Gerbong 3', out => "Data_block_1".sarana); END_IF;
   #_w16 := "Data_block_1"."counter" = 16;
   IF #_w16 AND "Data_block_1".ResetCounterDataSensor THEN
       "Data_block_1".dataroda1[15] := "Data_block_1".data_lama1;
       "Data_block_1".datasuhu1 := "Data_block_1".data_lama1;
   END_IF;
   IF #_w16 AND "Data_block_1".Lock_B THEN
       "Data_block_1".dataroda2[15] := "Data_block_1".data_lama2;
       "Data_block_1".datasuhu2 := "Data_block_1".data_lama2;
   END_IF;
   #_w17 := "Data_block_1"."counter" = 17;
   IF #_w17 AND "Data_block_1".ResetCounterDataSensor THEN
       "Data_block_1".dataroda1[16] := "Data_block_1".data_lama1;
       "Data_block_1".datasuhu1 := "Data_block_1".data_lama1;
   END_IF;
   IF #_w17 AND "Data_block_1".Lock_B THEN
       "Data_block_1".dataroda2[16] := "Data_block_1".data_lama2;
       "Data_block_1".datasuhu2 := "Data_block_1".data_lama2;
   END_IF;
   #_w18 := "Data_block_1"."counter" = 18;
   IF #_w18 AND "Data_block_1".ResetCounterDataSensor THEN
       "Data_block_1".dataroda1[17] := "Data_block_1".data_lama1;
       "Data_block_1".datasuhu1 := "Data_block_1".data_lama1;
   END_IF;
   IF #_w18 AND "Data_block_1".Lock_B THEN
       "Data_block_1".dataroda2[17] := "Data_block_1".data_lama2;
       "Data_block_1".datasuhu2 := "Data_block_1".data_lama2;
   END_IF;
   #_w19 := "Data_block_1"."counter" = 19;
   IF #_w19 AND "Data_block_1".ResetCounterDataSensor THEN
       "Data_block_1".dataroda1[18] := "Data_block_1".data_lama1;
       "Data_block_1".datasuhu1 := "Data_block_1".data_lama1;
   END_IF;
   IF #_w19 AND "Data_block_1".Lock_B THEN
       "Data_block_1".dataroda2[18] := "Data_block_1".data_lama2;
       "Data_block_1".datasuhu2 := "Data_block_1".data_lama2;
   END_IF;
   IF #_w19 THEN S_MOVE(in := 'Gerbong 4', out => "Data_block_1".sarana); END_IF;
   #_w20 := "Data_block_1"."counter" = 20;
   IF #_w20 AND "Data_block_1".ResetCounterDataSensor THEN
       "Data_block_1".dataroda1[19] := "Data_block_1".data_lama1;
       "Data_block_1".datasuhu1 := "Data_block_1".data_lama1;
   END_IF;
   IF #_w20 AND "Data_block_1".Lock_B THEN
       "Data_block_1".dataroda2[19] := "Data_block_1".data_lama2;
       "Data_block_1".datasuhu2 := "Data_block_1".data_lama2;
   END_IF;
   #_w21 := "Data_block_1"."counter" = 21;
   IF #_w21 AND "Data_block_1".ResetCounterDataSensor THEN
       "Data_block_1".dataroda1[20] := "Data_block_1".data_lama1;
       "Data_block_1".datasuhu1 := "Data_block_1".data_lama1;
   END_IF;
   IF #_w21 AND "Data_block_1".Lock_B THEN
       "Data_block_1".dataroda2[20] := "Data_block_1".data_lama2;
       "Data_block_1".datasuhu2 := "Data_block_1".data_lama2;
   END_IF;
   #_w22 := "Data_block_1"."counter" = 22;
   IF #_w22 AND "Data_block_1".ResetCounterDataSensor THEN
       "Data_block_1".dataroda1[21] := "Data_block_1".data_lama1;
       "Data_block_1".datasuhu1 := "Data_block_1".data_lama1;
   END_IF;
   IF #_w22 AND "Data_block_1".Lock_B THEN
       "Data_block_1".dataroda2[21] := "Data_block_1".data_lama2;
       "Data_block_1".datasuhu2 := "Data_block_1".data_lama2;
   END_IF;
   #_w23 := "Data_block_1"."counter" = 23;
   IF #_w23 AND "Data_block_1".ResetCounterDataSensor THEN
       "Data_block_1".dataroda1[22] := "Data_block_1".data_lama1;
       "Data_block_1".datasuhu1 := "Data_block_1".data_lama1;
   END_IF;
   IF #_w23 AND "Data_block_1".Lock_B THEN
       "Data_block_1".dataroda2[22] := "Data_block_1".data_lama2;
       "Data_block_1".datasuhu2 := "Data_block_1".data_lama2;
   END_IF;
   IF #_w23 THEN S_MOVE(in := 'Gerbong 5', out => "Data_block_1".sarana); END_IF;
   #_w24 := "Data_block_1"."counter" = 24;
   IF #_w24 AND "Data_block_1".ResetCounterDataSensor THEN
       "Data_block_1".dataroda1[23] := "Data_block_1".data_lama1;
       "Data_block_1".datasuhu1 := "Data_block_1".data_lama1;
   END_IF;
   IF #_w24 AND "Data_block_1".Lock_B THEN
       "Data_block_1".dataroda2[23] := "Data_block_1".data_lama2;
       "Data_block_1".datasuhu2 := "Data_block_1".data_lama2;
   END_IF;
   #_w25 := "Data_block_1"."counter" = 25;
   IF #_w25 AND "Data_block_1".ResetCounterDataSensor THEN
       "Data_block_1".dataroda1[24] := "Data_block_1".data_lama1;
       "Data_block_1".datasuhu1 := "Data_block_1".data_lama1;
   END_IF;
   IF #_w25 AND "Data_block_1".Lock_B THEN
       "Data_block_1".dataroda2[24] := "Data_block_1".data_lama2;
       "Data_block_1".datasuhu2 := "Data_block_1".data_lama2;
   END_IF;
   #_w26 := "Data_block_1"."counter" = 26;
   IF #_w26 AND "Data_block_1".ResetCounterDataSensor THEN
       "Data_block_1".dataroda1[25] := "Data_block_1".data_lama1;
       "Data_block_1".datasuhu1 := "Data_block_1".data_lama1;
   END_IF;
   IF #_w26 AND "Data_block_1".Lock_B THEN
       "Data_block_1".dataroda2[25] := "Data_block_1".data_lama2;
       "Data_block_1".datasuhu2 := "Data_block_1".data_lama2;
   END_IF;
   #_w27 := "Data_block_1"."counter" = 27;
   IF #_w27 AND "Data_block_1".ResetCounterDataSensor THEN
       "Data_block_1".dataroda1[26] := "Data_block_1".data_lama1;
       "Data_block_1".datasuhu1 := "Data_block_1".data_lama1;
   END_IF;
   IF #_w27 AND "Data_block_1".Lock_B THEN
       "Data_block_1".dataroda2[26] := "Data_block_1".data_lama2;
       "Data_block_1".datasuhu2 := "Data_block_1".data_lama2;
   END_IF;
   IF #_w27 THEN S_MOVE(in := 'Gerbong 6', out => "Data_block_1".sarana); END_IF;
   #_w28 := "Data_block_1"."counter" = 28;
   IF #_w28 AND "Data_block_1".ResetCounterDataSensor THEN
       "Data_block_1".dataroda1[27] := "Data_block_1".data_lama1;
       "Data_block_1".datasuhu1 := "Data_block_1".data_lama1;
   END_IF;
   IF #_w28 AND "Data_block_1".Lock_B THEN
       "Data_block_1".dataroda2[27] := "Data_block_1".data_lama2;
       "Data_block_1".datasuhu2 := "Data_block_1".data_lama2;
   END_IF;
   #_w29 := "Data_block_1"."counter" = 29;
   IF #_w29 AND "Data_block_1".ResetCounterDataSensor THEN
       "Data_block_1".dataroda1[28] := "Data_block_1".data_lama1;
       "Data_block_1".datasuhu1 := "Data_block_1".data_lama1;
   END_IF;
   IF #_w29 AND "Data_block_1".Lock_B THEN
       "Data_block_1".dataroda2[28] := "Data_block_1".data_lama2;
       "Data_block_1".datasuhu2 := "Data_block_1".data_lama2;
   END_IF;
   #_w30 := "Data_block_1"."counter" = 30;
   IF #_w30 AND "Data_block_1".ResetCounterDataSensor THEN
       "Data_block_1".dataroda1[29] := "Data_block_1".data_lama1;
       "Data_block_1".datasuhu1 := "Data_block_1".data_lama1;
   END_IF;
   IF #_w30 AND "Data_block_1".Lock_B THEN
       "Data_block_1".dataroda2[29] := "Data_block_1".data_lama2;
       "Data_block_1".datasuhu2 := "Data_block_1".data_lama2;
   END_IF;
   #_w31 := "Data_block_1"."counter" = 31;
   IF #_w31 AND "Data_block_1".ResetCounterDataSensor THEN
       "Data_block_1".dataroda1[30] := "Data_block_1".data_lama1;
       "Data_block_1".datasuhu1 := "Data_block_1".data_lama1;
   END_IF;
   IF #_w31 AND "Data_block_1".Lock_B THEN
       "Data_block_1".dataroda2[30] := "Data_block_1".data_lama2;
       "Data_block_1".datasuhu2 := "Data_block_1".data_lama2;
   END_IF;
   IF #_w31 THEN S_MOVE(in := 'Gerbong 7', out => "Data_block_1".sarana); END_IF;
   #_w32 := "Data_block_1"."counter" = 32;
   IF #_w32 AND "Data_block_1".ResetCounterDataSensor THEN
       "Data_block_1".dataroda1[31] := "Data_block_1".data_lama1;
       "Data_block_1".datasuhu1 := "Data_block_1".data_lama1;
   END_IF;
   IF #_w32 AND "Data_block_1".Lock_B THEN
       "Data_block_1".dataroda2[31] := "Data_block_1".data_lama2;
       "Data_block_1".datasuhu2 := "Data_block_1".data_lama2;
   END_IF;
   #_w33 := "Data_block_1"."counter" = 33;
   IF #_w33 AND "Data_block_1".ResetCounterDataSensor THEN
       "Data_block_1".dataroda1[32] := "Data_block_1".data_lama1;
       "Data_block_1".datasuhu1 := "Data_block_1".data_lama1;
   END_IF;
   IF #_w33 AND "Data_block_1".Lock_B THEN
       "Data_block_1".dataroda2[32] := "Data_block_1".data_lama2;
       "Data_block_1".datasuhu2 := "Data_block_1".data_lama2;
   END_IF;
   #_w34 := "Data_block_1"."counter" = 34;
   IF #_w34 AND "Data_block_1".ResetCounterDataSensor THEN
       "Data_block_1".dataroda1[33] := "Data_block_1".data_lama1;
       "Data_block_1".datasuhu1 := "Data_block_1".data_lama1;
   END_IF;
   IF #_w34 AND "Data_block_1".Lock_B THEN
       "Data_block_1".dataroda2[33] := "Data_block_1".data_lama2;
       "Data_block_1".datasuhu2 := "Data_block_1".data_lama2;
   END_IF;
   #_w35 := "Data_block_1"."counter" = 35;
   IF #_w35 AND "Data_block_1".ResetCounterDataSensor THEN
       "Data_block_1".dataroda1[34] := "Data_block_1".data_lama1;
       "Data_block_1".datasuhu1 := "Data_block_1".data_lama1;
   END_IF;
   IF #_w35 AND "Data_block_1".Lock_B THEN
       "Data_block_1".dataroda2[34] := "Data_block_1".data_lama2;
       "Data_block_1".datasuhu2 := "Data_block_1".data_lama2;
   END_IF;
   IF #_w35 THEN S_MOVE(in := 'Gerbong 8', out => "Data_block_1".sarana); END_IF;
   #_w36 := "Data_block_1"."counter" = 36;
   IF #_w36 AND "Data_block_1".ResetCounterDataSensor THEN
       "Data_block_1".dataroda1[35] := "Data_block_1".data_lama1;
       "Data_block_1".datasuhu1 := "Data_block_1".data_lama1;
   END_IF;
   IF #_w36 AND "Data_block_1".Lock_B THEN
       "Data_block_1".dataroda2[35] := "Data_block_1".data_lama2;
       "Data_block_1".datasuhu2 := "Data_block_1".data_lama2;
   END_IF;
   #_w37 := "Data_block_1"."counter" = 37;
   IF #_w37 AND "Data_block_1".ResetCounterDataSensor THEN
       "Data_block_1".dataroda1[36] := "Data_block_1".data_lama1;
       "Data_block_1".datasuhu1 := "Data_block_1".data_lama1;
   END_IF;
   IF #_w37 AND "Data_block_1".Lock_B THEN
       "Data_block_1".dataroda2[36] := "Data_block_1".data_lama2;
       "Data_block_1".datasuhu2 := "Data_block_1".data_lama2;
   END_IF;
   #_w38 := "Data_block_1"."counter" = 38;
   IF #_w38 AND "Data_block_1".ResetCounterDataSensor THEN
       "Data_block_1".dataroda1[37] := "Data_block_1".data_lama1;
       "Data_block_1".datasuhu1 := "Data_block_1".data_lama1;
   END_IF;
   IF #_w38 AND "Data_block_1".Lock_B THEN
       "Data_block_1".dataroda2[37] := "Data_block_1".data_lama2;
       "Data_block_1".datasuhu2 := "Data_block_1".data_lama2;
   END_IF;
   #_w39 := "Data_block_1"."counter" = 39;
   IF #_w39 AND "Data_block_1".ResetCounterDataSensor THEN
       "Data_block_1".dataroda1[38] := "Data_block_1".data_lama1;
       "Data_block_1".datasuhu1 := "Data_block_1".data_lama1;
   END_IF;
   IF #_w39 AND "Data_block_1".Lock_B THEN
       "Data_block_1".dataroda2[38] := "Data_block_1".data_lama2;
       "Data_block_1".datasuhu2 := "Data_block_1".data_lama2;
   END_IF;
   IF #_w39 THEN S_MOVE(in := 'Gerbong 9', out => "Data_block_1".sarana); END_IF;
   #_w40 := "Data_block_1"."counter" = 40;
   IF #_w40 AND "Data_block_1".ResetCounterDataSensor THEN
       "Data_block_1".dataroda1[39] := "Data_block_1".data_lama1;
       "Data_block_1".datasuhu1 := "Data_block_1".data_lama1;
   END_IF;
   IF #_w40 AND "Data_block_1".Lock_B THEN
       "Data_block_1".dataroda2[39] := "Data_block_1".data_lama2;
       "Data_block_1".datasuhu2 := "Data_block_1".data_lama2;
   END_IF;
   #_w41 := "Data_block_1"."counter" = 41;
   IF #_w41 AND "Data_block_1".ResetCounterDataSensor THEN
       "Data_block_1".dataroda1[40] := "Data_block_1".data_lama1;
       "Data_block_1".datasuhu1 := "Data_block_1".data_lama1;
   END_IF;
   IF #_w41 AND "Data_block_1".Lock_B THEN
       "Data_block_1".dataroda2[40] := "Data_block_1".data_lama2;
       "Data_block_1".datasuhu2 := "Data_block_1".data_lama2;
   END_IF;
   #_w42 := "Data_block_1"."counter" = 42;
   IF #_w42 AND "Data_block_1".ResetCounterDataSensor THEN
       "Data_block_1".dataroda1[41] := "Data_block_1".data_lama1;
       "Data_block_1".datasuhu1 := "Data_block_1".data_lama1;
   END_IF;
   IF #_w42 AND "Data_block_1".Lock_B THEN
       "Data_block_1".dataroda2[41] := "Data_block_1".data_lama2;
       "Data_block_1".datasuhu2 := "Data_block_1".data_lama2;
   END_IF;
   #_w43 := "Data_block_1"."counter" = 43;
   IF #_w43 AND "Data_block_1".ResetCounterDataSensor THEN
       "Data_block_1".dataroda1[42] := "Data_block_1".data_lama1;
       "Data_block_1".datasuhu1 := "Data_block_1".data_lama1;
   END_IF;
   IF #_w43 AND "Data_block_1".Lock_B THEN
       "Data_block_1".dataroda2[42] := "Data_block_1".data_lama2;
       "Data_block_1".datasuhu2 := "Data_block_1".data_lama2;
   END_IF;
   IF #_w43 THEN S_MOVE(in := 'Gerbong 10', out => "Data_block_1".sarana); END_IF;
   #_w44 := "Data_block_1"."counter" = 44;
   IF #_w44 AND "Data_block_1".ResetCounterDataSensor THEN
       "Data_block_1".dataroda1[43] := "Data_block_1".data_lama1;
       "Data_block_1".datasuhu1 := "Data_block_1".data_lama1;
   END_IF;
   IF #_w44 AND "Data_block_1".Lock_B THEN
       "Data_block_1".dataroda2[43] := "Data_block_1".data_lama2;
       "Data_block_1".datasuhu2 := "Data_block_1".data_lama2;
   END_IF;
   #_w45 := "Data_block_1"."counter" = 45;
   IF #_w45 AND "Data_block_1".ResetCounterDataSensor THEN
       "Data_block_1".dataroda1[44] := "Data_block_1".data_lama1;
       "Data_block_1".datasuhu1 := "Data_block_1".data_lama1;
   END_IF;
   IF #_w45 AND "Data_block_1".Lock_B THEN
       "Data_block_1".dataroda2[44] := "Data_block_1".data_lama2;
       "Data_block_1".datasuhu2 := "Data_block_1".data_lama2;
   END_IF;
   #_w46 := "Data_block_1"."counter" = 46;
   IF #_w46 AND "Data_block_1".ResetCounterDataSensor THEN
       "Data_block_1".dataroda1[45] := "Data_block_1".data_lama1;
       "Data_block_1".datasuhu1 := "Data_block_1".data_lama1;
   END_IF;
   IF #_w46 AND "Data_block_1".Lock_B THEN
       "Data_block_1".dataroda2[45] := "Data_block_1".data_lama2;
       "Data_block_1".datasuhu2 := "Data_block_1".data_lama2;
   END_IF;
   #_w47 := "Data_block_1"."counter" = 47;
   IF #_w47 AND "Data_block_1".ResetCounterDataSensor THEN
       "Data_block_1".dataroda1[46] := "Data_block_1".data_lama1;
       "Data_block_1".datasuhu1 := "Data_block_1".data_lama1;
   END_IF;
   IF #_w47 AND "Data_block_1".Lock_B THEN
       "Data_block_1".dataroda2[46] := "Data_block_1".data_lama2;
       "Data_block_1".datasuhu2 := "Data_block_1".data_lama2;
   END_IF;
   IF #_w47 THEN S_MOVE(in := 'Gerbong11', out => "Data_block_1".sarana); END_IF;
   #_w48 := "Data_block_1"."counter" = 48;
   IF #_w48 AND "Data_block_1".ResetCounterDataSensor THEN
       "Data_block_1".dataroda1[47] := "Data_block_1".data_lama1;
       "Data_block_1".datasuhu1 := "Data_block_1".data_lama1;
   END_IF;
   IF #_w48 AND "Data_block_1".Lock_B THEN
       "Data_block_1".dataroda2[47] := "Data_block_1".data_lama2;
       "Data_block_1".datasuhu2 := "Data_block_1".data_lama2;
   END_IF;
   #_w49 := "Data_block_1"."counter" = 49;
   IF #_w49 AND "Data_block_1".ResetCounterDataSensor THEN
       "Data_block_1".dataroda1[48] := "Data_block_1".data_lama1;
       "Data_block_1".datasuhu1 := "Data_block_1".data_lama1;
   END_IF;
   IF #_w49 AND "Data_block_1".Lock_B THEN
       "Data_block_1".dataroda2[48] := "Data_block_1".data_lama2;
       "Data_block_1".datasuhu2 := "Data_block_1".data_lama2;
   END_IF;
   #_w50 := "Data_block_1"."counter" = 50;
   IF #_w50 AND "Data_block_1".ResetCounterDataSensor THEN
       "Data_block_1".dataroda1[49] := "Data_block_1".data_lama1;
       "Data_block_1".datasuhu1 := "Data_block_1".data_lama1;
   END_IF;
   IF #_w50 AND "Data_block_1".Lock_B THEN
       "Data_block_1".dataroda2[49] := "Data_block_1".data_lama2;
       "Data_block_1".datasuhu2 := "Data_block_1".data_lama2;
   END_IF;
END_REGION

REGION Network 30: Koil Reset
   // ketika sensor prox a tidak aktif selama 30 detik, reset akan aktif
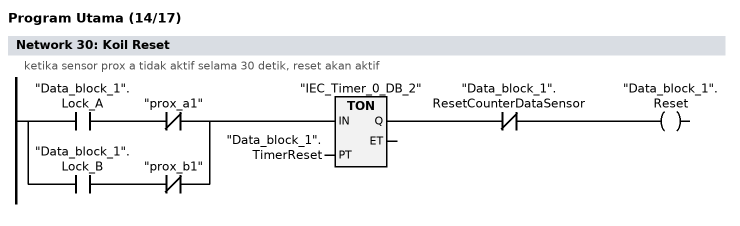
   "IEC_Timer_0_DB_2".TON(IN := ("Data_block_1".Lock_A AND NOT "prox_a1") OR ("Data_block_1".Lock_B AND NOT "prox_b1"),
                          PT := "Data_block_1".TimerReset);
   "Data_block_1".Reset := "IEC_Timer_0_DB_2".Q AND NOT "Data_block_1".ResetCounterDataSensor;
END_REGION

REGION Network 31: reset data suhu roda
   // ketika reset aktif 
   // 
   // - maka datasuhu, array data suhu roda akan kembali 0
   // - maka counter genap kembali 0
   // - maka counter ganjil menjadi -1
   // - maka sarana akan kosong
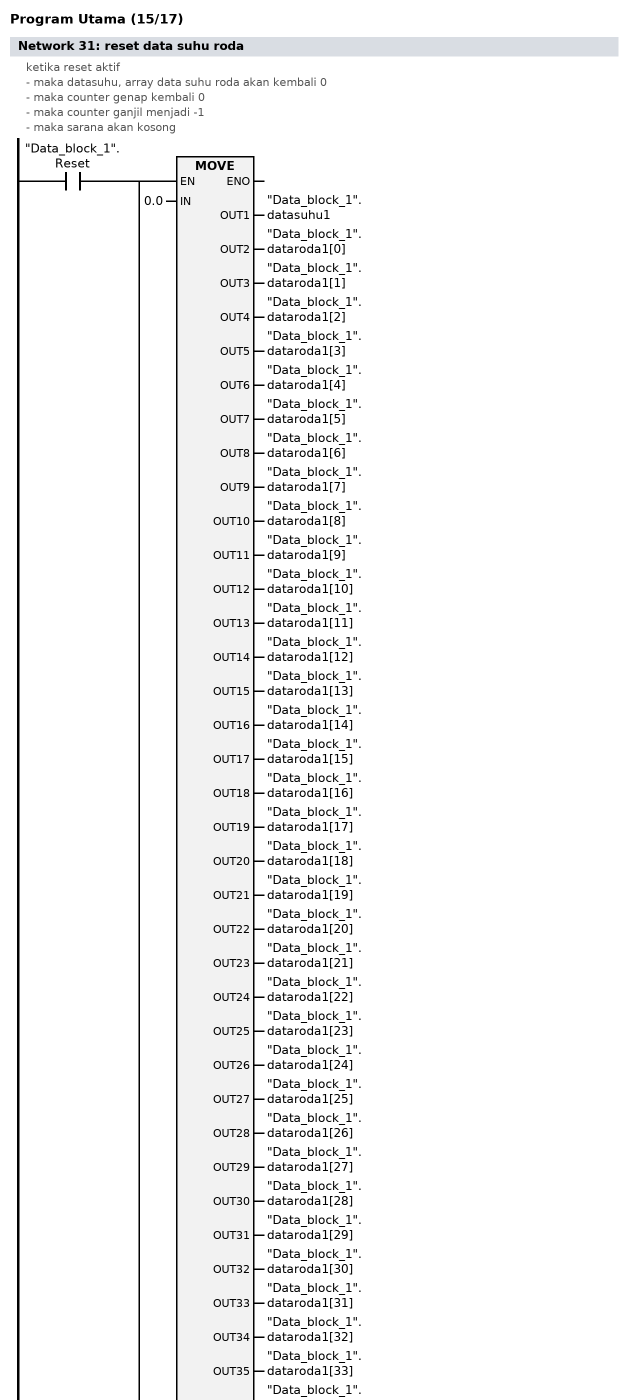
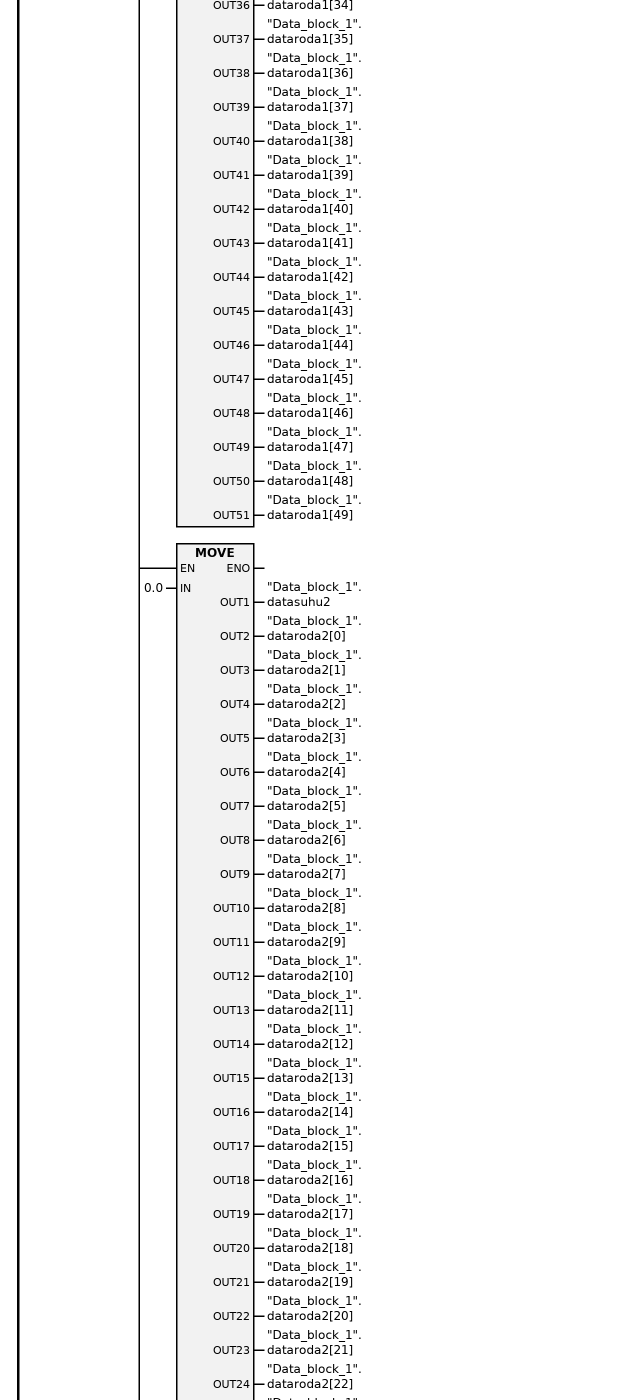
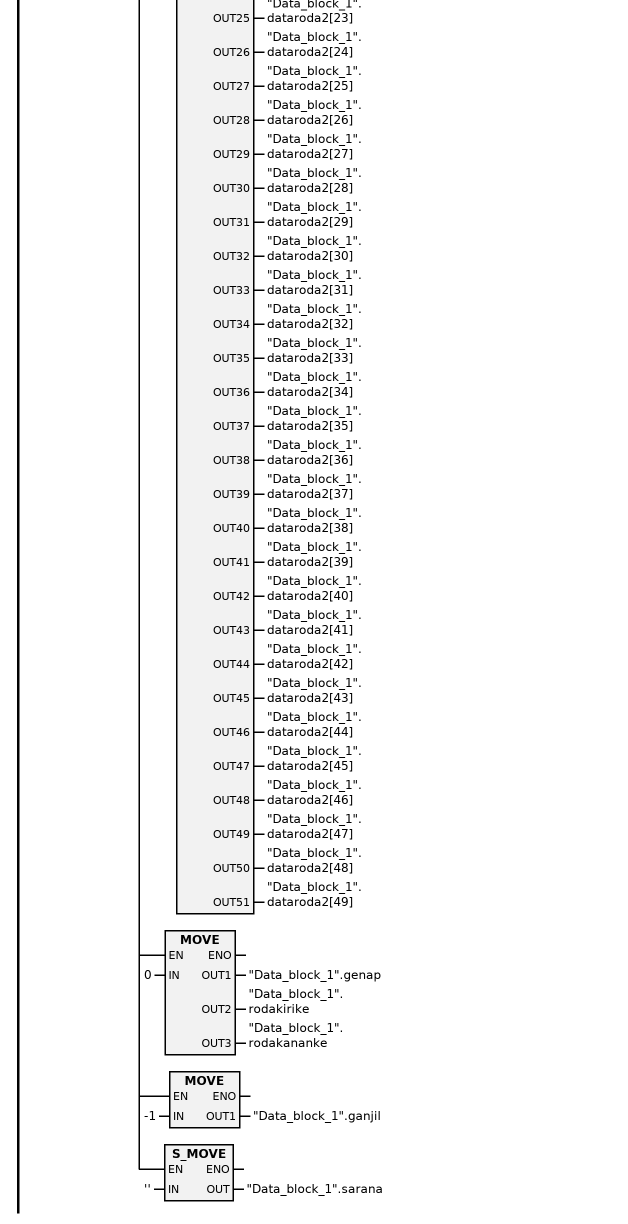
   IF "Data_block_1".Reset THEN
       "Data_block_1".datasuhu1 := 0.0;
       "Data_block_1".dataroda1[0] := 0.0;
       "Data_block_1".dataroda1[1] := 0.0;
       "Data_block_1".dataroda1[2] := 0.0;
       "Data_block_1".dataroda1[3] := 0.0;
       "Data_block_1".dataroda1[4] := 0.0;
       "Data_block_1".dataroda1[5] := 0.0;
       "Data_block_1".dataroda1[6] := 0.0;
       "Data_block_1".dataroda1[7] := 0.0;
       "Data_block_1".dataroda1[8] := 0.0;
       "Data_block_1".dataroda1[9] := 0.0;
       "Data_block_1".dataroda1[10] := 0.0;
       "Data_block_1".dataroda1[11] := 0.0;
       "Data_block_1".dataroda1[12] := 0.0;
       "Data_block_1".dataroda1[13] := 0.0;
       "Data_block_1".dataroda1[14] := 0.0;
       "Data_block_1".dataroda1[15] := 0.0;
       "Data_block_1".dataroda1[16] := 0.0;
       "Data_block_1".dataroda1[17] := 0.0;
       "Data_block_1".dataroda1[18] := 0.0;
       "Data_block_1".dataroda1[19] := 0.0;
       "Data_block_1".dataroda1[20] := 0.0;
       "Data_block_1".dataroda1[21] := 0.0;
       "Data_block_1".dataroda1[22] := 0.0;
       "Data_block_1".dataroda1[23] := 0.0;
       "Data_block_1".dataroda1[24] := 0.0;
       "Data_block_1".dataroda1[25] := 0.0;
       "Data_block_1".dataroda1[26] := 0.0;
       "Data_block_1".dataroda1[27] := 0.0;
       "Data_block_1".dataroda1[28] := 0.0;
       "Data_block_1".dataroda1[29] := 0.0;
       "Data_block_1".dataroda1[30] := 0.0;
       "Data_block_1".dataroda1[31] := 0.0;
       "Data_block_1".dataroda1[32] := 0.0;
       "Data_block_1".dataroda1[33] := 0.0;
       "Data_block_1".dataroda1[34] := 0.0;
       "Data_block_1".dataroda1[35] := 0.0;
       "Data_block_1".dataroda1[36] := 0.0;
       "Data_block_1".dataroda1[37] := 0.0;
       "Data_block_1".dataroda1[38] := 0.0;
       "Data_block_1".dataroda1[39] := 0.0;
       "Data_block_1".dataroda1[40] := 0.0;
       "Data_block_1".dataroda1[41] := 0.0;
       "Data_block_1".dataroda1[42] := 0.0;
       "Data_block_1".dataroda1[43] := 0.0;
       "Data_block_1".dataroda1[44] := 0.0;
       "Data_block_1".dataroda1[45] := 0.0;
       "Data_block_1".dataroda1[46] := 0.0;
       "Data_block_1".dataroda1[47] := 0.0;
       "Data_block_1".dataroda1[48] := 0.0;
       "Data_block_1".dataroda1[49] := 0.0;
       "Data_block_1".datasuhu2 := 0.0;
       "Data_block_1".dataroda2[0] := 0.0;
       "Data_block_1".dataroda2[1] := 0.0;
       "Data_block_1".dataroda2[2] := 0.0;
       "Data_block_1".dataroda2[3] := 0.0;
       "Data_block_1".dataroda2[4] := 0.0;
       "Data_block_1".dataroda2[5] := 0.0;
       "Data_block_1".dataroda2[6] := 0.0;
       "Data_block_1".dataroda2[7] := 0.0;
       "Data_block_1".dataroda2[8] := 0.0;
       "Data_block_1".dataroda2[9] := 0.0;
       "Data_block_1".dataroda2[10] := 0.0;
       "Data_block_1".dataroda2[11] := 0.0;
       "Data_block_1".dataroda2[12] := 0.0;
       "Data_block_1".dataroda2[13] := 0.0;
       "Data_block_1".dataroda2[14] := 0.0;
       "Data_block_1".dataroda2[15] := 0.0;
       "Data_block_1".dataroda2[16] := 0.0;
       "Data_block_1".dataroda2[17] := 0.0;
       "Data_block_1".dataroda2[18] := 0.0;
       "Data_block_1".dataroda2[19] := 0.0;
       "Data_block_1".dataroda2[20] := 0.0;
       "Data_block_1".dataroda2[21] := 0.0;
       "Data_block_1".dataroda2[22] := 0.0;
       "Data_block_1".dataroda2[23] := 0.0;
       "Data_block_1".dataroda2[24] := 0.0;
       "Data_block_1".dataroda2[25] := 0.0;
       "Data_block_1".dataroda2[26] := 0.0;
       "Data_block_1".dataroda2[27] := 0.0;
       "Data_block_1".dataroda2[28] := 0.0;
       "Data_block_1".dataroda2[29] := 0.0;
       "Data_block_1".dataroda2[30] := 0.0;
       "Data_block_1".dataroda2[31] := 0.0;
       "Data_block_1".dataroda2[32] := 0.0;
       "Data_block_1".dataroda2[33] := 0.0;
       "Data_block_1".dataroda2[34] := 0.0;
       "Data_block_1".dataroda2[35] := 0.0;
       "Data_block_1".dataroda2[36] := 0.0;
       "Data_block_1".dataroda2[37] := 0.0;
       "Data_block_1".dataroda2[38] := 0.0;
       "Data_block_1".dataroda2[39] := 0.0;
       "Data_block_1".dataroda2[40] := 0.0;
       "Data_block_1".dataroda2[41] := 0.0;
       "Data_block_1".dataroda2[42] := 0.0;
       "Data_block_1".dataroda2[43] := 0.0;
       "Data_block_1".dataroda2[44] := 0.0;
       "Data_block_1".dataroda2[45] := 0.0;
       "Data_block_1".dataroda2[46] := 0.0;
       "Data_block_1".dataroda2[47] := 0.0;
       "Data_block_1".dataroda2[48] := 0.0;
       "Data_block_1".dataroda2[49] := 0.0;
       "Data_block_1".genap := 0;
       "Data_block_1".rodakirike := 0;
       "Data_block_1".rodakananke := 0;
       "Data_block_1".ganjil := -1;
       S_MOVE(in := '', out => "Data_block_1".sarana);
   END_IF;
END_REGION

REGION Network 32: running led
   // program running led penunjuk arah
